C01820=1061.242,135.759,420.443,172.181,30.453,155.636
C01821=1061.248,136.008,420.422,172.183,30.455,155.637
C01822=1061.253,136.258,420.401,172.185,30.458,155.637
C01823=1061.259,136.507,420.381,172.186,30.461,155.638
C01824=1061.266,136.756,420.359,172.188,30.463,155.638
C01825=1061.271,137.005,420.339,172.190,30.466,155.638
C01826=1061.278,137.254,420.318,172.192,30.469,155.639
C01827=1061.283,137.503,420.297,172.193,30.471,155.639
C01828=1061.289,137.751,420.276,172.195,30.474,155.640
C01829=1061.295,138.001,420.255,172.197,30.477,155.640
C01830=1061.300,138.250,420.235,172.199,30.480,155.640
C01831=1061.307,138.499,420.213,172.201,30.482,155.641
C01832=1061.313,138.748,420.193,172.202,30.485,155.641
C01833=1061.319,138.997,420.172,172.204,30.488,155.642
C01834=1061.324,139.246,420.151,172.205,30.490,155.642
C01835=1061.331,139.495,420.130,172.207,30.493,155.643
C01836=1061.336,139.744,420.109,172.208,30.495,155.643
C01837=1061.342,139.993,420.088,172.210,30.498,155.643
C01838=1061.348,140.243,420.067,172.212,30.501,155.644
C01839=1061.353,140.491,420.046,172.214,30.503,155.644
C01840=1061.360,140.741,420.026,172.215,30.507,155.645
C01841=1061.365,140.989,420.004,172.217,30.509,155.645
C01842=1061.371,141.239,419.983,172.219,30.512,155.646
C01843=1061.377,141.488,419.962,172.221,30.515,155.646
C01844=1061.383,141.737,419.941,172.223,30.517,155.646
C01845=1061.388,141.986,419.920,172.224,30.520,155.647
C01846=1061.395,142.270,419.896,172.226,30.523,155.647
C01847=1061.402,142.554,419.872,172.229,30.526,155.648
C01848=1061.409,142.839,419.848,172.231,30.529,155.648
C01849=1061.416,143.123,419.824,172.232,30.533,155.649
C01850=1061.421,143.372,419.803,172.234,30.535,155.649
C01851=1061.427,143.621,419.781,172.236,30.538,155.650
C01852=1061.433,143.870,419.760,172.238,30.541,155.650
C01853=1061.438,144.120,419.739,172.239,30.543,155.650
C01854=1061.444,144.368,419.718,172.241,30.546,155.651
C01855=1061.450,144.617,419.696,172.243,30.549,155.651
C01856=1061.455,144.866,419.676,172.245,30.551,155.652
C01857=1061.462,145.115,419.655,172.246,30.554,155.652
C01858=1061.468,145.364,419.633,172.248,30.557,155.653
C01859=1061.474,145.613,419.612,172.250,30.560,155.653
C01860=1061.480,145.863,419.591,172.252,30.563,155.653
C01861=1061.486,146.111,419.570,172.254,30.565,155.654
C01862=1061.492,146.361,419.548,172.255,30.568,155.654
C01863=1061.497,146.610,419.527,172.257,30.571,155.655
C01864=1061.503,146.859,419.506,172.259,30.573,155.655
C01865=1061.509,147.107,419.485,172.261,30.576,155.655
C01866=1061.515,147.357,419.463,172.262,30.579,155.656
C01867=1061.522,147.605,419.442,172.264,30.581,155.656
C01868=1061.527,147.855,419.421,172.266,30.584,155.657
C01869=1061.532,148.104,419.399,172.268,30.587,155.657
C01870=1061.538,148.353,419.378,172.270,30.590,155.658
C01871=1061.544,148.602,419.356,172.271,30.592,155.658
C01872=1061.550,148.850,419.335,172.273,30.595,155.658
C01873=1061.556,149.100,419.313,172.275,30.598,155.659
C01874=1061.562,149.349,419.292,172.277,30.600,155.659
C01875=1061.567,149.598,419.271,172.278,30.603,155.660
C01876=1061.573,149.847,419.249,172.280,30.606,155.660
C01877=1061.579,150.096,419.228,172.282,30.609,155.661
C01878=1061.585,150.345,419.207,172.284,30.612,155.661
C01879=1061.591,150.594,419.185,172.286,30.614,155.662
C01880=1061.597,150.843,419.164,172.287,30.617,155.662
C01881=1061.603,151.092,419.142,172.289,30.620,155.662
C01882=1061.608,151.341,419.120,172.291,30.622,155.663
C01883=1061.614,151.590,419.099,172.294,30.625,155.663
C01884=1061.620,151.839,419.077,172.295,30.628,155.664
C01885=1061.626,152.087,419.056,172.297,30.631,155.664
C01886=1061.632,152.337,419.034,172.299,30.634,155.665
C01887=1061.637,152.585,419.013,172.301,30.636,155.665
C01888=1061.644,152.834,418.991,172.302,30.639,155.665
C01889=1061.649,153.084,418.969,172.304,30.642,155.666
C01890=1061.655,153.332,418.948,172.306,30.645,155.666
C01891=1061.661,153.582,418.926,172.308,30.648,155.667
C01892=1061.667,153.831,418.904,172.310,30.650,155.667
C01893=1061.673,154.079,418.883,172.311,30.653,155.668
C01894=1061.679,154.329,418.861,172.313,30.656,155.668
C01895=1061.684,154.578,418.839,172.315,30.658,155.668
C01896=1061.690,154.827,418.818,172.317,30.661,155.669
C01897=1061.696,155.076,418.796,172.318,30.664,155.669
C01898=1061.702,155.325,418.775,172.320,30.667,155.670
C01899=1061.708,155.573,418.753,172.322,30.669,155.670
C01900=1061.713,155.822,418.730,172.324,30.672,155.671
C01901=1061.719,156.072,418.709,172.326,30.675,155.671
C01902=1061.726,156.321,418.687,172.327,30.678,155.671
C01903=1061.730,156.570,418.665,172.330,30.681,155.672
C01904=1061.737,156.819,418.644,172.332,30.684,155.672
C01905=1061.743,157.068,418.622,172.334,30.686,155.673
C01906=1061.748,157.316,418.599,172.336,30.689,155.673
C01907=1061.754,157.565,418.578,172.337,30.692,155.674
C01908=1061.760,157.815,418.556,172.339,30.695,155.674
C01909=1061.766,158.063,418.535,172.341,30.697,155.675
C01910=1061.773,158.348,418.509,172.343,30.701,155.675
C01911=1061.779,158.631,418.484,172.345,30.704,155.676
C01912=1061.786,158.915,418.460,172.347,30.707,155.676
C01913=1061.793,159.200,418.434,172.349,30.710,155.676
C01914=1061.798,159.448,418.413,172.351,30.713,155.677
C01915=1061.804,159.698,418.391,172.353,30.716,155.677
C01916=1061.810,159.946,418.368,172.355,30.719,155.678
C01917=1061.816,160.196,418.347,172.357,30.721,155.678
C01918=1061.821,160.444,418.325,172.359,30.724,155.679
C01919=1061.827,160.693,418.303,172.361,30.727,155.679
C01920=1061.834,160.942,418.281,172.362,30.729,155.679
C01921=1061.839,161.192,418.259,172.364,30.732,155.680
C01922=1061.845,161.440,418.237,172.366,30.735,155.680
C01923=1061.850,161.689,418.214,172.368,30.738,155.681
C01924=1061.856,161.938,418.191,172.369,30.741,155.681
C01925=1061.862,162.187,418.170,172.371,30.744,155.682
C01926=1061.867,162.436,418.148,172.374,30.747,155.682
C01927=1061.873,162.685,418.125,172.376,30.750,155.683
C01928=1061.879,162.934,418.103,172.378,30.752,155.683
C01929=1061.884,163.182,418.081,172.379,30.756,155.684
C01930=1061.889,163.432,418.059,172.381,30.758,155.684
C01931=1061.896,163.680,418.036,172.383,30.761,155.685
C01932=1061.901,163.930,418.014,172.385,30.764,155.685
C01933=1061.907,164.178,417.991,172.386,30.767,155.685
C01934=1061.913,164.427,417.970,172.388,30.770,155.686
C01935=1061.918,164.676,417.947,172.390,30.773,155.686
C01936=1061.924,164.926,417.925,172.393,30.775,155.687
C01937=1061.929,165.174,417.902,172.395,30.779,155.687
C01938=1061.935,165.423,417.880,172.396,30.781,155.688
C01939=1061.941,165.672,417.857,172.398,30.785,155.688
C01940=1061.946,165.922,417.835,172.400,30.787,155.689
C01941=1061.952,166.169,417.813,172.402,30.790,155.689
C01942=1061.958,166.419,417.791,172.403,30.793,155.690
C01943=1061.963,166.668,417.768,172.405,30.796,155.690
C01944=1061.970,166.916,417.746,172.407,30.798,155.691
C01945=1061.975,167.166,417.723,172.410,30.802,155.691
C01946=1061.981,167.415,417.701,172.412,30.804,155.691
C01947=1061.986,167.664,417.679,172.413,30.808,155.692
C01948=1061.992,167.912,417.656,172.415,30.810,155.692
C01949=1061.998,168.161,417.633,172.417,30.813,155.693
C01950=1062.003,168.411,417.611,172.419,30.816,155.693
C01951=1062.009,168.660,417.588,172.421,30.819,155.694
C01952=1062.016,168.908,417.566,172.423,30.822,155.694
C01953=1062.020,169.157,417.544,172.425,30.825,155.695
C01954=1062.026,169.406,417.521,172.427,30.827,155.695
C01955=1062.033,169.654,417.499,172.429,30.830,155.696
C01956=1062.038,169.904,417.476,172.430,30.833,155.696
C01957=1062.044,170.153,417.454,172.432,30.836,155.696
C01958=1062.049,170.402,417.431,172.434,30.839,155.697
C01959=1062.055,170.651,417.408,172.437,30.842,155.697
C01960=1062.061,170.900,417.386,172.439,30.845,155.698
C01961=1062.067,171.148,417.363,172.440,30.848,155.698
C01962=1062.072,171.397,417.340,172.442,30.850,155.699
C01963=1062.078,171.646,417.318,172.444,30.853,155.699
C01964=1062.084,171.895,417.296,172.446,30.856,155.700
C01965=1062.090,172.144,417.273,172.448,30.859,155.700
C01966=1062.096,172.393,417.250,172.450,30.862,155.701
C01967=1062.101,172.642,417.227,172.452,30.865,155.701
C01968=1062.108,172.890,417.205,172.454,30.868,155.702
C01969=1062.113,173.140,417.182,172.456,30.871,155.702
C01970=1062.119,173.389,417.160,172.457,30.874,155.702
C01971=1062.125,173.638,417.137,172.460,30.876,155.703
C01972=1062.130,173.887,417.114,172.462,30.880,155.703
C01973=1062.137,174.135,417.091,172.464,30.882,155.704
C01974=1062.143,174.419,417.066,172.467,30.886,155.704
C01975=1062.150,174.703,417.040,172.468,30.889,155.705
C01976=1062.156,174.986,417.013,172.471,30.892,155.705
C01977=1062.163,175.270,416.988,172.473,30.895,155.706
C01978=1062.169,175.518,416.965,172.475,30.898,155.706
C01979=1062.175,175.767,416.942,172.476,30.901,155.707
C01980=1062.180,176.016,416.919,172.479,30.904,155.707
C01981=1062.186,176.265,416.896,172.481,30.907,155.708
C01982=1062.192,176.514,416.874,172.483,30.910,155.708
C01983=1062.198,176.763,416.851,172.485,30.912,155.709
C01984=1062.204,177.012,416.828,172.486,30.915,155.709
C01985=1062.210,177.261,416.805,172.489,30.919,155.710
C01986=1062.216,177.510,416.782,172.491,30.921,155.710
C01987=1062.222,177.759,416.759,172.493,30.924,155.710
C01988=1062.228,178.008,416.736,172.495,30.927,155.711
C01989=1062.233,178.257,416.713,172.497,30.930,155.711
C01990=1062.240,178.505,416.691,172.499,30.932,155.712
C01991=1062.246,178.754,416.668,172.501,30.936,155.712
C01992=1062.251,179.003,416.645,172.503,30.938,155.713
C01993=1062.257,179.252,416.622,172.505,30.941,155.713
C01994=1062.263,179.501,416.599,172.507,30.944,155.714
C01995=1062.269,179.749,416.575,172.509,30.947,155.714
C01996=1062.275,179.998,416.553,172.511,30.950,155.715
C01997=1062.282,180.247,416.530,172.513,30.953,155.715
C01998=1062.287,180.496,416.507,172.516,30.956,155.715
C01999=1062.293,180.745,416.484,172.517,30.959,155.716
C02000=1062.299,180.994,416.461,172.519,30.961,155.716
C02001=1062.305,181.243,416.438,172.521,30.964,155.717
C02002=1062.311,181.491,416.414,172.524,30.967,155.717
C02003=1062.316,181.740,416.391,172.525,30.970,155.718
C02004=1062.323,181.989,416.369,172.527,30.973,155.718
C02005=1062.329,182.238,416.346,172.529,30.976,155.719
C02006=1062.335,182.487,416.323,172.532,30.979,155.719
C02007=1062.341,182.735,416.299,172.534,30.981,155.720
C02008=1062.347,182.984,416.276,172.535,30.984,155.720
C02009=1062.353,183.234,416.253,172.538,30.987,155.720
C02010=1062.359,183.483,416.230,172.540,30.990,155.721
C02011=1062.364,183.732,416.207,172.542,30.993,155.721
C02012=1062.370,183.980,416.183,172.544,30.996,155.722
C02013=1062.376,184.229,416.160,172.546,30.999,155.722
C02014=1062.383,184.478,416.138,172.548,31.002,155.723
C02015=1062.389,184.727,416.113,172.550,31.005,155.723
C02016=1062.394,184.976,416.090,172.552,31.008,155.724
C02017=1062.399,185.225,416.067,172.555,31.011,155.724
C02018=1062.405,185.473,416.043,172.556,31.014,155.725
C02019=1062.411,185.722,416.020,172.558,31.017,155.725
C02020=1062.416,185.971,415.996,172.561,31.020,155.726
C02021=1062.422,186.220,415.973,172.563,31.023,155.726
C02022=1062.428,186.469,415.950,172.565,31.026,155.727
C02023=1062.434,186.718,415.925,172.566,31.029,155.727
C02024=1062.439,186.967,415.902,172.569,31.032,155.728
C02025=1062.445,187.215,415.879,172.571,31.035,155.728
C02026=1062.450,187.464,415.855,172.573,31.038,155.729
C02027=1062.456,187.712,415.832,172.575,31.041,155.729
C02028=1062.461,187.962,415.808,172.577,31.044,155.730
C02029=1062.468,188.211,415.784,172.579,31.048,155.730
C02030=1062.474,188.459,415.761,172.581,31.050,155.731
C02031=1062.479,188.708,415.737,172.584,31.053,155.731
C02032=1062.485,188.957,415.714,172.585,31.057,155.732
C02033=1062.490,189.206,415.690,172.587,31.059,155.732
C02034=1062.496,189.454,415.667,172.590,31.063,155.733
C02035=1062.503,189.703,415.643,172.592,31.066,155.733
C02036=1062.508,189.952,415.618,172.594,31.068,155.734
C02037=1062.514,190.201,415.595,172.595,31.072,155.734
C02038=1062.520,190.484,415.568,172.598,31.075,155.735
C02039=1062.527,190.768,415.542,172.601,31.079,155.735
C02040=1062.533,191.050,415.514,172.603,31.082,155.736
C02041=1062.540,191.334,415.487,172.606,31.086,155.736
C02042=1062.546,191.583,415.464,172.607,31.089,155.737
C02043=1062.551,191.831,415.439,172.610,31.091,155.737
C02044=1062.557,192.080,415.416,172.612,31.095,155.738
C02045=1062.563,192.329,415.392,172.614,31.098,155.738
C02046=1062.569,192.578,415.368,172.617,31.101,155.739
C02047=1062.575,192.826,415.345,172.618,31.104,155.739
C02048=1062.580,193.075,415.321,172.620,31.107,155.740
C02049=1062.586,193.324,415.297,172.623,31.110,155.740
C02050=1062.591,193.573,415.273,172.625,31.113,155.741
C02051=1062.597,193.822,415.250,172.627,31.116,155.741
C02052=1062.603,194.071,415.225,172.629,31.120,155.742
C02053=1062.609,194.319,415.202,172.631,31.122,155.742
C02054=1062.615,194.568,415.178,172.633,31.125,155.743
C02055=1062.621,194.817,415.153,172.636,31.129,155.743
C02056=1062.627,195.066,415.130,172.638,31.131,155.744
C02057=1062.632,195.314,415.106,172.639,31.135,155.744
C02058=1062.639,195.563,415.082,172.642,31.138,155.745
C02059=1062.644,195.812,415.058,172.644,31.140,155.745
C02060=1062.650,196.060,415.034,172.647,31.144,155.746
C02061=1062.656,196.310,415.010,172.649,31.147,155.746
C02062=1062.662,196.558,414.987,172.650,31.150,155.747
C02063=1062.668,196.808,414.962,172.653,31.153,155.747
C02064=1062.674,197.056,414.938,172.655,31.156,155.748
C02065=1062.679,197.305,414.914,172.657,31.159,155.748
C02066=1062.686,197.554,414.890,172.660,31.162,155.749
C02067=1062.691,197.802,414.866,172.661,31.165,155.749
C02068=1062.697,198.050,414.842,172.664,31.169,155.750
C02069=1062.703,198.300,414.817,172.666,31.171,155.750
C02070=1062.709,198.548,414.794,172.668,31.174,155.751
C02071=1062.714,198.798,414.770,172.671,31.178,155.751
C02072=1062.720,199.046,414.746,172.672,31.180,155.752
C02073=1062.726,199.295,414.722,172.675,31.184,155.752
C02074=1062.732,199.544,414.698,172.677,31.187,155.753
C02075=1062.738,199.793,414.673,172.679,31.190,155.753
C02076=1062.744,200.041,414.650,172.682,31.193,155.754
C02077=1062.750,200.290,414.625,172.683,31.196,155.754
C02078=1062.756,200.539,414.601,172.686,31.199,155.755
C02079=1062.762,200.787,414.576,172.688,31.202,155.755
C02080=1062.768,201.036,414.552,172.690,31.205,155.756
C02081=1062.774,201.284,414.528,172.693,31.209,155.756
C02082=1062.780,201.534,414.503,172.694,31.211,155.757
C02083=1062.786,201.782,414.480,172.697,31.214,155.757
C02084=1062.792,202.031,414.455,172.699,31.218,155.758
C02085=1062.797,202.280,414.431,172.702,31.221,155.758
C02086=1062.804,202.529,414.407,172.704,31.224,155.759
C02087=1062.809,202.777,414.383,172.705,31.227,155.759
C02088=1062.815,203.026,414.357,172.708,31.230,155.760
C02089=1062.820,203.275,414.333,172.710,31.233,155.760
C02090=1062.826,203.524,414.308,172.713,31.237,155.761
C02091=1062.832,203.772,414.285,172.715,31.240,155.761
C02092=1062.838,204.021,414.260,172.717,31.243,155.762
C02093=1062.844,204.269,414.235,172.719,31.246,155.763
C02094=1062.850,204.519,414.211,172.721,31.250,155.763
C02095=1062.855,204.767,414.186,172.724,31.253,155.764
C02096=1062.861,205.017,414.162,172.726,31.256,155.764
C02097=1062.867,205.264,414.137,172.728,31.259,155.765
C02098=1062.873,205.514,414.113,172.730,31.262,155.765
C02099=1062.879,205.762,414.088,172.733,31.265,155.766
C02100=1062.884,206.011,414.064,172.735,31.268,155.766
C02101=1062.890,206.259,414.039,172.738,31.272,155.767
C02102=1062.915,207.308,413.935,172.906,31.353,155.774
C02103=1062.920,207.532,413.912,172.908,31.357,155.775
C02104=1062.926,207.757,413.890,172.910,31.361,155.775
C02105=1062.931,207.982,413.866,172.911,31.364,155.776
C02106=1062.937,208.207,413.844,172.913,31.368,155.777
C02107=1062.943,208.432,413.821,172.915,31.372,155.777
C02108=1062.948,208.657,413.797,172.917,31.376,155.778
C02109=1062.953,208.881,413.775,172.919,31.379,155.779
C02110=1062.959,209.107,413.752,172.920,31.383,155.779
C02111=1062.965,209.355,413.726,172.922,31.387,155.780
C02112=1062.971,209.604,413.700,172.924,31.391,155.781
C02113=1062.977,209.852,413.674,172.926,31.395,155.782
C02114=1062.983,210.101,413.649,172.928,31.399,155.782
C02115=1062.989,210.350,413.624,172.930,31.404,155.783
C02116=1062.996,210.598,413.598,172.932,31.407,155.784
C02117=1063.001,210.847,413.572,172.934,31.412,155.784
C02118=1063.008,211.095,413.546,172.936,31.415,155.785
C02119=1063.014,211.344,413.521,172.937,31.420,155.786
C02120=1063.019,211.593,413.495,172.939,31.423,155.787
C02121=1063.025,211.842,413.470,172.942,31.428,155.787
C02122=1063.032,212.090,413.444,172.944,31.432,155.788
C02123=1063.038,212.338,413.418,172.946,31.436,155.789
C02124=1063.044,212.587,413.392,172.947,31.440,155.790
C02125=1063.050,212.836,413.367,172.949,31.444,155.790
C02126=1063.055,213.085,413.341,172.952,31.448,155.791
C02127=1063.062,213.333,413.315,172.954,31.452,155.792
C02128=1063.068,213.582,413.290,172.956,31.456,155.792
C02129=1063.073,213.831,413.264,172.957,31.460,155.793
C02130=1063.080,214.079,413.238,172.959,31.464,155.794
C02131=1063.085,214.328,413.212,172.962,31.469,155.795
C02132=1063.092,214.576,413.186,172.964,31.472,155.795
C02133=1063.097,214.825,413.160,172.966,31.477,155.796
C02134=1063.104,215.073,413.134,172.967,31.480,155.797
C02135=1063.109,215.322,413.108,172.969,31.485,155.798
C02136=1063.116,215.570,413.082,172.972,31.488,155.798
C02137=1063.122,215.819,413.057,172.974,31.493,155.799
C02138=1063.128,216.068,413.031,172.976,31.496,155.800
C02139=1063.134,216.316,413.005,172.977,31.501,155.801
C02140=1063.140,216.565,412.979,172.979,31.504,155.801
C02141=1063.146,216.813,412.953,172.982,31.509,155.802
C02142=1063.152,217.062,412.927,172.984,31.513,155.803
C02143=1063.158,217.310,412.901,172.986,31.517,155.803
C02144=1063.164,217.559,412.875,172.987,31.521,155.804
C02145=1063.170,217.808,412.849,172.990,31.525,155.805
C02146=1063.176,218.056,412.822,172.992,31.529,155.806
C02147=1063.182,218.305,412.797,172.994,31.533,155.806
C02148=1063.188,218.553,412.770,172.996,31.537,155.807
C02149=1063.194,218.802,412.745,172.998,31.541,155.808
C02150=1063.200,219.050,412.718,173.000,31.545,155.808
C02151=1063.206,219.299,412.693,173.002,31.549,155.809
C02152=1063.212,219.547,412.666,173.004,31.553,155.810
C02153=1063.219,219.797,412.641,173.007,31.557,155.811
C02154=1063.225,220.045,412.614,173.008,31.561,155.811
C02155=1063.231,220.293,412.588,173.010,31.565,155.812
C02156=1063.237,220.542,412.562,173.012,31.569,155.813
C02157=1063.243,220.790,412.536,173.015,31.573,155.813
C02158=1063.249,221.039,412.509,173.017,31.577,155.814
C02159=1063.254,221.266,412.485,173.019,31.581,155.815
C02160=1063.260,221.494,412.461,173.020,31.584,155.815
C02161=1063.265,221.721,412.438,173.022,31.588,155.816
C02162=1063.271,221.948,412.413,173.024,31.591,155.817
C02163=1063.277,222.176,412.389,173.026,31.595,155.817
C02164=1063.282,222.403,412.365,173.028,31.599,155.818
C02165=1063.288,222.630,412.341,173.030,31.602,155.819
C02166=1063.293,222.858,412.317,173.031,31.606,155.820
C02167=1063.299,223.106,412.290,173.034,31.611,155.820
C02168=1063.305,223.355,412.264,173.036,31.614,155.821
C02169=1063.310,223.603,412.237,173.038,31.619,155.822
C02170=1063.318,223.852,412.211,173.041,31.622,155.822
C02171=1063.323,224.100,412.184,173.042,31.627,155.823
C02172=1063.329,224.349,412.158,173.044,31.630,155.824
C02173=1063.335,224.598,412.132,173.046,31.635,155.825
C02174=1063.341,224.846,412.106,173.049,31.638,155.825
C02175=1063.347,225.095,412.079,173.051,31.642,155.826
C02176=1063.353,225.343,412.052,173.053,31.646,155.827
C02177=1063.359,225.592,412.025,173.055,31.650,155.827
C02178=1063.365,225.840,411.999,173.057,31.655,155.828
C02179=1063.372,226.089,411.972,173.059,31.658,155.829
C02180=1063.378,226.337,411.946,173.061,31.662,155.830
C02181=1063.383,226.585,411.919,173.064,31.666,155.830
C02182=1063.389,226.834,411.892,173.066,31.670,155.831
C02183=1063.395,227.084,411.866,173.067,31.674,155.832
C02184=1063.402,227.332,411.840,173.070,31.678,155.832
C02185=1063.408,227.580,411.813,173.072,31.682,155.833
C02186=1063.414,227.829,411.786,173.074,31.686,155.834
C02187=1063.420,228.077,411.760,173.077,31.690,155.835
C02188=1063.425,228.326,411.733,173.078,31.694,155.835
C02189=1063.433,228.574,411.707,173.080,31.698,155.836
C02190=1063.439,228.822,411.679,173.083,31.702,155.837
C02191=1063.444,229.071,411.653,173.085,31.706,155.838
C02192=1063.451,229.320,411.626,173.087,31.710,155.838
C02193=1063.457,229.568,411.599,173.090,31.714,155.839
C02194=1063.462,229.816,411.572,173.091,31.718,155.840
C02195=1063.469,230.065,411.545,173.093,31.721,155.840
C02196=1063.475,230.314,411.519,173.096,31.726,155.841
C02197=1063.480,230.562,411.492,173.098,31.730,155.842
C02198=1063.487,230.811,411.465,173.100,31.734,155.843
C02199=1063.492,231.060,411.438,173.103,31.738,155.843
C02200=1063.499,231.307,411.411,173.104,31.742,155.844
C02201=1063.505,231.556,411.384,173.106,31.746,155.845
C02202=1063.511,231.805,411.357,173.109,31.749,155.845
C02203=1063.516,232.053,411.331,173.111,31.754,155.846
C02204=1063.523,232.302,411.304,173.113,31.757,155.847
C02205=1063.529,232.550,411.276,173.116,31.762,155.848
C02206=1063.535,232.798,411.250,173.117,31.765,155.848
C02207=1063.541,233.047,411.223,173.119,31.770,155.849
C02208=1063.547,233.296,411.196,173.122,31.774,155.850
C02209=1063.553,233.544,411.168,173.124,31.777,155.850
C02210=1063.559,233.792,411.142,173.127,31.782,155.851
C02211=1063.564,234.041,411.114,173.129,31.785,155.852
C02212=1063.571,234.290,411.087,173.131,31.790,155.853
C02213=1063.577,234.538,411.060,173.133,31.793,155.853
C02214=1063.583,234.786,411.033,173.135,31.798,155.854
C02215=1063.588,235.010,411.009,173.137,31.801,155.855
C02216=1063.594,235.233,410.984,173.139,31.804,155.855
C02217=1063.599,235.457,410.960,173.141,31.808,155.856
C02218=1063.605,235.680,410.936,173.144,31.812,155.857
C02219=1063.610,235.903,410.911,173.146,31.815,155.857
C02220=1063.616,236.127,410.887,173.147,31.819,155.858
C02221=1063.621,236.350,410.862,173.149,31.822,155.859
C02222=1063.626,236.574,410.837,173.151,31.826,155.859
C02223=1063.632,236.821,410.810,173.154,31.830,155.860
C02224=1063.638,237.070,410.783,173.156,31.834,155.861
C02225=1063.644,237.318,410.756,173.158,31.838,155.861
C02226=1063.651,237.567,410.729,173.160,31.842,155.862
C02227=1063.657,237.815,410.701,173.162,31.846,155.863
C02228=1063.662,238.064,410.674,173.165,31.850,155.864
C02229=1063.669,238.312,410.646,173.167,31.853,155.864
C02230=1063.675,238.561,410.619,173.169,31.858,155.865
C02231=1063.681,238.809,410.592,173.172,31.861,155.866
C02232=1063.687,239.058,410.563,173.174,31.865,155.866
C02233=1063.693,239.306,410.537,173.176,31.869,155.867
C02234=1063.699,239.554,410.509,173.178,31.873,155.868
C02235=1063.705,239.803,410.482,173.180,31.877,155.868
C02236=1063.711,240.052,410.454,173.183,31.881,155.869
C02237=1063.717,240.299,410.427,173.185,31.885,155.870
C02238=1063.724,240.548,410.400,173.188,31.889,155.871
C02239=1063.729,240.796,410.372,173.190,31.893,155.871
C02240=1063.736,241.045,410.344,173.192,31.897,155.872
C02241=1063.742,241.294,410.317,173.194,31.900,155.873
C02242=1063.748,241.542,410.290,173.197,31.905,155.874
C02243=1063.754,241.790,410.261,173.199,31.908,155.874
C02244=1063.760,242.039,410.235,173.201,31.912,155.875
C02245=1063.766,242.287,410.207,173.204,31.917,155.876
C02246=1063.772,242.535,410.179,173.206,31.920,155.876
C02247=1063.778,242.784,410.151,173.208,31.925,155.877
C02248=1063.784,243.033,410.124,173.210,31.928,155.878
C02249=1063.790,243.281,410.096,173.213,31.932,155.878
C02250=1063.796,243.530,410.068,173.215,31.936,155.879
C02251=1063.802,243.777,410.041,173.218,31.940,155.880
C02252=1063.808,244.026,410.012,173.220,31.944,155.881
C02253=1063.814,244.274,409.986,173.222,31.948,155.881
C02254=1063.820,244.523,409.957,173.224,31.952,155.882
C02255=1063.827,244.772,409.930,173.226,31.956,155.883
C02256=1063.832,245.020,409.902,173.229,31.960,155.884
C02257=1063.839,245.268,409.874,173.231,31.964,155.884
C02258=1063.844,245.516,409.846,173.234,31.968,155.885
C02259=1063.851,245.765,409.818,173.236,31.972,155.886
C02260=1063.857,246.013,409.790,173.239,31.976,155.886
C02261=1063.862,246.261,409.762,173.241,31.980,155.887
C02262=1063.869,246.510,409.734,173.243,31.984,155.888
C02263=1063.874,246.758,409.706,173.245,31.988,155.889
C02264=1063.880,247.007,409.678,173.248,31.992,155.889
C02265=1063.886,247.255,409.650,173.250,31.996,155.890
C02266=1063.892,247.503,409.622,173.253,32.000,155.891
C02267=1063.898,247.752,409.594,173.255,32.004,155.892
C02268=1063.904,248.000,409.567,173.257,32.007,155.892
C02269=1063.910,248.248,409.538,173.259,32.012,155.893
C02270=1063.916,248.497,409.510,173.261,32.015,155.894
C02271=1063.921,248.717,409.485,173.264,32.019,155.894
C02272=1063.926,248.937,409.460,173.266,32.023,155.895
C02273=1063.932,249.157,409.435,173.268,32.026,155.896
C02274=1063.937,249.378,409.410,173.270,32.030,155.896
C02275=1063.942,249.598,409.386,173.272,32.033,155.897
C02276=1063.947,249.818,409.360,173.275,32.037,155.898
C02277=1063.953,250.038,409.336,173.277,32.040,155.898
C02278=1063.957,250.259,409.311,173.278,32.044,155.899
C02279=1063.964,250.507,409.282,173.281,32.048,155.900
C02280=1063.970,250.755,409.254,173.283,32.052,155.900
C02281=1063.976,251.003,409.226,173.286,32.056,155.901
C02282=1063.982,251.252,409.198,173.288,32.060,155.902
C02283=1063.988,251.500,409.168,173.291,32.064,155.902
C02284=1063.993,251.748,409.141,173.293,32.068,155.903
C02285=1064.000,251.997,409.113,173.296,32.072,155.904
C02286=1064.006,252.246,409.084,173.297,32.076,155.905
C02287=1064.012,252.493,409.056,173.300,32.080,155.905
C02288=1064.017,252.742,409.027,173.302,32.083,155.906
C02289=1064.023,252.991,408.999,173.305,32.088,155.907
C02290=1064.030,253.238,408.971,173.307,32.091,155.908
C02291=1064.036,253.487,408.942,173.310,32.096,155.908
C02292=1064.042,253.735,408.914,173.312,32.099,155.909
C02293=1064.048,253.983,408.885,173.315,32.103,155.910
C02294=1064.054,254.232,408.857,173.317,32.107,155.911
C02295=1064.060,254.481,408.829,173.319,32.111,155.911
C02296=1064.066,254.728,408.801,173.322,32.115,155.912
C02297=1064.072,254.977,408.772,173.324,32.119,155.913
C02298=1064.078,255.225,408.743,173.327,32.123,155.913
C02299=1064.084,255.474,408.715,173.329,32.127,155.914
C02300=1064.091,255.722,408.686,173.332,32.131,155.915
C02301=1064.097,255.970,408.658,173.335,32.135,155.915
C02302=1064.102,256.218,408.629,173.337,32.139,155.916
C02303=1064.109,256.466,408.601,173.339,32.143,155.917
C02304=1064.115,256.714,408.572,173.341,32.146,155.918
C02305=1064.121,256.963,408.544,173.344,32.151,155.918
C02306=1064.127,257.211,408.515,173.346,32.154,155.919
C02307=1064.133,257.460,408.486,173.349,32.158,155.920
C02308=1064.140,257.708,408.457,173.352,32.162,155.921
C02309=1064.145,257.957,408.429,173.354,32.166,155.921
C02310=1064.151,258.204,408.400,173.357,32.170,155.922
C02311=1064.158,258.453,408.373,173.359,32.174,155.923
C02312=1064.164,258.701,408.344,173.361,32.178,155.923
C02313=1064.170,258.949,408.315,173.364,32.181,155.924
C02314=1064.176,259.198,408.286,173.366,32.186,155.925
C02315=1064.182,259.446,408.257,173.369,32.189,155.926
C02316=1064.189,259.694,408.228,173.371,32.193,155.926
C02317=1064.195,259.943,408.200,173.374,32.197,155.927
C02318=1064.201,260.191,408.171,173.377,32.201,155.928
C02319=1064.207,260.439,408.142,173.379,32.205,155.928
C02320=1064.213,260.688,408.113,173.382,32.209,155.929
C02321=1064.220,260.936,408.085,173.384,32.213,155.930
C02322=1064.226,261.184,408.056,173.386,32.217,155.931
C02323=1064.233,261.432,408.027,173.389,32.220,155.931
C02324=1064.239,261.681,407.999,173.391,32.225,155.932
C02325=1064.245,261.929,407.970,173.394,32.228,155.933
C02326=1064.251,262.177,407.941,173.397,32.232,155.933
C02327=1064.257,262.397,407.915,173.399,32.236,155.934
C02328=1064.262,262.615,407.889,173.401,32.239,155.935
C02329=1064.267,262.835,407.864,173.404,32.243,155.935
C02330=1064.273,263.053,407.839,173.406,32.246,155.936
C02331=1064.278,263.273,407.813,173.408,32.249,155.937
C02332=1064.284,263.492,407.787,173.410,32.252,155.937
C02333=1064.289,263.711,407.762,173.412,32.256,155.938
C02334=1064.295,263.930,407.736,173.414,32.260,155.938
C02335=1064.301,264.178,407.707,173.417,32.263,155.939
C02336=1064.307,264.426,407.678,173.420,32.268,155.940
C02337=1064.313,264.675,407.648,173.422,32.271,155.941
C02338=1064.319,264.923,407.619,173.425,32.276,155.941
C02339=1064.325,265.171,407.590,173.428,32.280,155.942
C02340=1064.332,265.419,407.561,173.430,32.283,155.943
C02341=1064.337,265.668,407.531,173.433,32.287,155.944
C02342=1064.343,265.916,407.502,173.436,32.291,155.944
C02343=1064.350,266.164,407.473,173.437,32.295,155.945
C02344=1064.356,266.412,407.444,173.440,32.299,155.946
C02345=1064.361,266.660,407.414,173.443,32.303,155.946
C02346=1064.368,266.908,407.385,173.445,32.307,155.947
C02347=1064.374,267.157,407.356,173.448,32.311,155.948
C02348=1064.379,267.405,407.327,173.451,32.315,155.949
C02349=1064.386,267.653,407.298,173.453,32.319,155.949
C02350=1064.392,267.901,407.269,173.456,32.323,155.950
C02351=1064.398,268.149,407.238,173.459,32.327,155.951
C02352=1064.404,268.397,407.209,173.461,32.331,155.952
C02353=1064.410,268.645,407.180,173.464,32.335,155.952
C02354=1064.417,268.894,407.151,173.466,32.339,155.953
C02355=1064.422,269.143,407.121,173.468,32.343,155.954
C02356=1064.429,269.391,407.092,173.471,32.347,155.954
C02357=1064.435,269.639,407.062,173.474,32.351,155.955
C02358=1064.441,269.887,407.033,173.476,32.354,155.956
C02359=1064.446,270.135,407.003,173.479,32.359,155.957
C02360=1064.453,270.383,406.973,173.482,32.363,155.957
C02361=1064.459,270.631,406.944,173.485,32.367,155.958
C02362=1064.465,270.879,406.915,173.487,32.370,155.959
C02363=1064.472,271.128,406.885,173.490,32.375,155.960
C02364=1064.477,271.376,406.855,173.493,32.378,155.960
C02365=1064.484,271.624,406.826,173.495,32.382,155.961
C02366=1064.489,271.872,406.796,173.497,32.386,155.962
C02367=1064.496,272.120,406.767,173.500,32.390,155.963
C02368=1064.501,272.368,406.737,173.503,32.394,155.963
C02369=1064.508,272.617,406.707,173.505,32.398,155.964
C02370=1064.514,272.865,406.677,173.508,32.402,155.965
C02371=1064.520,273.113,406.647,173.511,32.406,155.965
C02372=1064.526,273.361,406.618,173.513,32.410,155.966
C02373=1064.532,273.609,406.588,173.516,32.414,155.967
C02374=1064.538,273.857,406.558,173.519,32.418,155.968
C02375=1064.545,274.105,406.528,173.522,32.422,155.968
C02376=1064.551,274.354,406.499,173.524,32.426,155.969
C02377=1064.556,274.602,406.468,173.527,32.430,155.970
C02378=1064.563,274.850,406.439,173.530,32.434,155.971
C02379=1064.568,275.097,406.409,173.532,32.438,155.971
C02380=1064.575,275.347,406.379,173.534,32.442,155.972
C02381=1064.581,275.594,406.349,173.537,32.446,155.973
C02382=1064.587,275.842,406.319,173.540,32.450,155.974
C02383=1064.593,276.063,406.293,173.542,32.454,155.974
C02384=1064.598,276.284,406.266,173.545,32.458,155.975
C02385=1064.603,276.505,406.239,173.547,32.461,155.976
C02386=1064.609,276.726,406.213,173.550,32.464,155.976
C02387=1064.614,276.947,406.186,173.552,32.468,155.977
C02388=1064.620,277.168,406.158,173.555,32.472,155.978
C02389=1064.625,277.388,406.132,173.557,32.475,155.978
C02390=1064.630,277.609,406.105,173.560,32.479,155.979
C02391=1064.637,277.858,406.075,173.562,32.483,155.980
C02392=1064.643,278.106,406.046,173.565,32.487,155.981
C02393=1064.649,278.354,406.015,173.568,32.491,155.981
C02394=1064.655,278.602,405.985,173.570,32.495,155.982
C02395=1064.662,278.850,405.955,173.572,32.499,155.983
C02396=1064.667,279.098,405.925,173.575,32.503,155.983
C02397=1064.674,279.347,405.894,173.578,32.507,155.984
C02398=1064.679,279.595,405.864,173.581,32.511,155.985
C02399=1064.686,279.842,405.834,173.584,32.515,155.986
C02400=1064.692,280.091,405.804,173.586,32.519,155.986
C02401=1064.698,280.338,405.773,173.589,32.523,155.987
C02402=1064.704,280.586,405.743,173.592,32.527,155.988
C02403=1064.710,280.835,405.713,173.595,32.531,155.989
C02404=1064.716,281.083,405.683,173.598,32.535,155.989
C02405=1064.722,281.331,405.652,173.600,32.539,155.990
C02406=1064.728,281.580,405.621,173.603,32.543,155.991
C02407=1064.735,281.827,405.592,173.606,32.547,155.992
C02408=1064.741,282.075,405.561,173.609,32.551,155.993
C02409=1064.747,282.323,405.531,173.612,32.556,155.993
C02410=1064.753,282.571,405.500,173.615,32.559,155.994
C02411=1064.759,282.819,405.470,173.616,32.563,155.995
C02412=1064.765,283.068,405.439,173.619,32.568,155.996
C02413=1064.771,283.315,405.409,173.622,32.571,155.996
C02414=1064.777,283.563,405.378,173.625,32.576,155.997
C02415=1064.783,283.811,405.347,173.628,32.579,155.998
C02416=1064.789,284.059,405.317,173.631,32.584,155.999
C02417=1064.796,284.307,405.286,173.633,32.588,155.999
C02418=1064.801,284.555,405.256,173.636,32.592,156.000
C02419=1064.807,284.803,405.225,173.639,32.596,156.001
C02420=1064.814,285.052,405.195,173.642,32.600,156.002
C02421=1064.819,285.299,405.164,173.645,32.604,156.002
C02422=1064.826,285.547,405.133,173.648,32.608,156.003
C02423=1064.832,285.795,405.102,173.650,32.612,156.004
C02424=1064.838,286.044,405.072,173.653,32.616,156.005
C02425=1064.844,286.292,405.041,173.656,32.620,156.005
C02426=1064.851,286.539,405.010,173.659,32.624,156.006
C02427=1064.857,286.787,404.980,173.662,32.628,156.007
C02428=1064.863,287.036,404.949,173.665,32.632,156.008
C02429=1064.869,287.284,404.919,173.668,32.636,156.008
C02430=1064.876,287.531,404.887,173.670,32.640,156.009
C02431=1064.882,287.779,404.857,173.672,32.645,156.010
C02432=1064.888,288.028,404.826,173.675,32.648,156.011
C02433=1064.894,288.275,404.795,173.678,32.653,156.012
C02434=1064.901,288.524,404.764,173.681,32.657,156.012
C02435=1064.906,288.771,404.734,173.684,32.661,156.013
C02436=1064.913,289.019,404.702,173.687,32.665,156.014
C02437=1064.918,289.267,404.672,173.690,32.669,156.015
C02438=1064.925,289.515,404.640,173.693,32.673,156.015
C02439=1064.931,289.742,404.612,173.695,32.677,156.016
C02440=1064.936,289.967,404.584,173.698,32.681,156.017
C02441=1064.942,290.194,404.556,173.701,32.684,156.018
C02442=1064.948,290.420,404.527,173.703,32.688,156.018
C02443=1064.953,290.646,404.499,173.706,32.692,156.019
C02444=1064.959,290.872,404.471,173.709,32.696,156.020
C02445=1064.965,291.099,404.443,173.711,32.699,156.020
C02446=1064.970,291.325,404.414,173.714,32.703,156.021
C02447=1064.976,291.572,404.383,173.717,32.707,156.022
C02448=1064.982,291.821,404.352,173.720,32.711,156.023
C02449=1064.988,292.068,404.321,173.723,32.715,156.023
C02450=1064.994,292.316,404.289,173.726,32.720,156.024
C02451=1065.001,292.565,404.258,173.729,32.724,156.025
C02452=1065.007,292.812,404.227,173.731,32.728,156.026
C02453=1065.013,293.061,404.196,173.734,32.732,156.027
C02454=1065.019,293.308,404.165,173.737,32.736,156.027
C02455=1065.025,293.556,404.133,173.740,32.740,156.028
C02456=1065.032,293.804,404.102,173.743,32.744,156.029
C02457=1065.037,294.052,404.071,173.745,32.749,156.030
C02458=1065.044,294.300,404.040,173.748,32.752,156.030
C02459=1065.051,294.548,404.008,173.751,32.757,156.031
C02460=1065.056,294.796,403.977,173.754,32.761,156.032
C02461=1065.062,295.044,403.946,173.757,32.765,156.033
C02462=1065.068,295.292,403.914,173.760,32.769,156.034
C02463=1065.075,295.539,403.883,173.763,32.773,156.034
C02464=1065.081,295.787,403.851,173.766,32.777,156.035
C02465=1065.087,296.035,403.819,173.769,32.782,156.036
C02466=1065.093,296.283,403.789,173.772,32.786,156.037
C02467=1065.099,296.531,403.757,173.775,32.790,156.038
C02468=1065.106,296.779,403.725,173.778,32.794,156.038
C02469=1065.111,297.027,403.694,173.781,32.799,156.039
C02470=1065.118,297.275,403.662,173.784,32.803,156.040
C02471=1065.124,297.523,403.630,173.787,32.807,156.041
C02472=1065.130,297.770,403.599,173.790,32.811,156.042
C02473=1065.136,298.018,403.567,173.793,32.815,156.042
C02474=1065.142,298.267,403.535,173.796,32.820,156.043
C02475=1065.147,298.514,403.503,173.799,32.824,156.044
C02476=1065.154,298.762,403.472,173.802,32.828,156.045
C02477=1065.160,299.010,403.440,173.805,32.832,156.046
C02478=1065.165,299.258,403.408,173.808,32.837,156.046
C02479=1065.172,299.506,403.377,173.811,32.841,156.047
C02480=1065.178,299.754,403.345,173.814,32.845,156.048
C02481=1065.184,300.001,403.312,173.817,32.849,156.049
C02482=1065.190,300.249,403.280,173.820,32.854,156.050
C02483=1065.197,300.497,403.249,173.823,32.858,156.051
C02484=1065.203,300.745,403.217,173.826,32.862,156.051
C02485=1065.208,300.993,403.185,173.829,32.866,156.052
C02486=1065.214,301.241,403.153,173.832,32.871,156.053
C02487=1065.221,301.488,403.121,173.835,32.875,156.054
C02488=1065.227,301.736,403.089,173.838,32.880,156.055
C02489=1065.233,301.985,403.057,173.841,32.884,156.056
C02490=1065.238,302.232,403.025,173.844,32.888,156.056
C02491=1065.245,302.479,402.993,173.847,32.892,156.057
C02492=1065.251,302.728,402.961,173.850,32.896,156.058
C02493=1065.257,302.976,402.929,173.853,32.901,156.059
C02494=1065.264,303.223,402.896,173.856,32.905,156.060
C02495=1065.269,303.457,402.867,173.859,32.909,156.060
C02496=1065.275,303.690,402.837,173.862,32.913,156.061
C02497=1065.281,303.924,402.807,173.865,32.917,156.062
C02498=1065.286,304.158,402.776,173.867,32.921,156.063
C02499=1065.293,304.391,402.746,173.870,32.925,156.064
C02500=1065.298,304.625,402.715,173.873,32.929,156.064
C02501=1065.304,304.859,402.685,173.876,32.933,156.065
C02502=1065.310,305.093,402.655,173.879,32.937,156.066
C02503=1065.316,305.341,402.622,173.882,32.942,156.067
C02504=1065.323,305.588,402.591,173.885,32.946,156.068
C02505=1065.329,305.836,402.558,173.888,32.950,156.068
C02506=1065.335,306.084,402.526,173.891,32.954,156.069
C02507=1065.341,306.332,402.493,173.894,32.959,156.070
C02508=1065.347,306.580,402.461,173.897,32.963,156.071
C02509=1065.354,306.827,402.429,173.901,32.968,156.072
C02510=1065.360,307.076,402.397,173.904,32.972,156.073
C02511=1065.366,307.322,402.364,173.907,32.976,156.073
C02512=1065.372,307.571,402.332,173.910,32.980,156.074
C02513=1065.378,307.818,402.300,173.913,32.985,156.075
C02514=1065.385,308.066,402.267,173.916,32.989,156.076
C02515=1065.391,308.314,402.235,173.919,32.993,156.077
C02516=1065.398,308.561,402.203,173.922,32.998,156.078
C02517=1065.404,308.809,402.170,173.925,33.002,156.078
C02518=1065.411,309.058,402.138,173.929,33.006,156.079
C02519=1065.417,309.305,402.105,173.932,33.010,156.080
C02520=1065.423,309.553,402.072,173.935,33.015,156.081
C02521=1065.429,309.801,402.040,173.938,33.019,156.082
C02522=1065.435,310.049,402.007,173.941,33.024,156.083
C02523=1065.442,310.296,401.975,173.944,33.028,156.083
C02524=1065.449,310.544,401.943,173.947,33.032,156.084
C02525=1065.455,310.791,401.910,173.951,33.036,156.085
C02526=1065.461,311.039,401.878,173.954,33.041,156.086
C02527=1065.467,311.287,401.845,173.957,33.045,156.087
C02528=1065.474,311.535,401.812,173.960,33.049,156.088
C02529=1065.480,311.782,401.780,173.963,33.054,156.088
C02530=1065.487,312.031,401.746,173.966,33.058,156.089
C02531=1065.493,312.278,401.714,173.970,33.062,156.090
C02532=1065.499,312.526,401.682,173.973,33.067,156.091
C02533=1065.505,312.774,401.649,173.976,33.071,156.092
C02534=1065.512,313.022,401.616,173.979,33.075,156.093
C02535=1065.519,313.269,401.584,173.982,33.080,156.093
C02536=1065.526,313.517,401.551,173.985,33.084,156.094
C02537=1065.532,313.765,401.518,173.989,33.089,156.095
C02538=1065.538,314.012,401.485,173.992,33.093,156.096
C02539=1065.544,314.260,401.452,173.995,33.098,156.097
C02540=1065.550,314.508,401.419,173.998,33.102,156.098
C02541=1065.556,314.755,401.387,174.001,33.106,156.099
C02542=1065.562,315.003,401.353,174.004,33.111,156.099
C02543=1065.568,315.250,401.320,174.008,33.116,156.100
C02544=1065.575,315.499,401.286,174.011,33.120,156.101
C02545=1065.581,315.746,401.253,174.014,33.124,156.102
C02546=1065.586,315.994,401.220,174.017,33.129,156.103
C02547=1065.593,316.242,401.187,174.020,33.133,156.104
C02548=1065.599,316.489,401.154,174.023,33.138,156.105
C02549=1065.605,316.737,401.120,174.027,33.142,156.106
C02550=1065.612,316.985,401.087,174.031,33.147,156.107
C02551=1065.618,317.224,401.055,174.034,33.151,156.107
C02552=1065.623,317.463,401.022,174.037,33.156,156.108
C02553=1065.629,317.702,400.991,174.040,33.160,156.109
C02554=1065.635,317.942,400.959,174.043,33.164,156.110
C02555=1065.641,318.180,400.927,174.046,33.169,156.111
C02556=1065.648,318.419,400.895,174.049,33.173,156.112
C02557=1065.653,318.658,400.862,174.053,33.178,156.113
C02558=1065.659,318.897,400.830,174.056,33.182,156.114
C02559=1065.665,319.141,400.797,174.059,33.187,156.114
C02560=1065.672,319.386,400.764,174.062,33.191,156.115
C02561=1065.677,319.630,400.732,174.065,33.195,156.116
C02562=1065.683,319.874,400.698,174.068,33.200,156.117
C02563=1065.689,320.118,400.665,174.072,33.205,156.118
C02564=1065.696,320.363,400.632,174.075,33.209,156.119
C02565=1065.702,320.607,400.599,174.078,33.214,156.120
C02566=1065.708,320.850,400.566,174.081,33.218,156.121
C02567=1065.714,321.098,400.533,174.084,33.223,156.122
C02568=1065.721,321.346,400.499,174.088,33.228,156.123
C02569=1065.727,321.593,400.465,174.091,33.232,156.123
C02570=1065.733,321.841,400.432,174.094,33.237,156.124
C02571=1065.740,322.089,400.398,174.097,33.241,156.125
C02572=1065.746,322.336,400.365,174.101,33.246,156.126
C02573=1065.752,322.584,400.331,174.105,33.250,156.127
C02574=1065.759,322.832,400.298,174.108,33.255,156.128
C02575=1065.765,323.079,400.264,174.111,33.260,156.129
C02576=1065.772,323.327,400.230,174.115,33.264,156.130
C02577=1065.777,323.575,400.197,174.118,33.269,156.131
C02578=1065.785,323.823,400.163,174.121,33.273,156.132
C02579=1065.790,324.070,400.129,174.125,33.278,156.133
C02580=1065.797,324.318,400.095,174.128,33.282,156.133
C02581=1065.803,324.565,400.062,174.131,33.287,156.134
C02582=1065.809,324.813,400.028,174.135,33.292,156.135
C02583=1065.816,325.060,399.994,174.138,33.297,156.136
C02584=1065.822,325.308,399.960,174.141,33.301,156.137
C02585=1065.829,325.556,399.927,174.144,33.306,156.138
C02586=1065.835,325.803,399.893,174.148,33.310,156.139
C02587=1065.841,326.051,399.858,174.151,33.315,156.140
C02588=1065.848,326.299,399.824,174.154,33.320,156.141
C02589=1065.854,326.546,399.790,174.158,33.325,156.142
C02590=1065.862,326.794,399.757,174.162,33.329,156.143
C02591=1065.867,327.041,399.723,174.165,33.333,156.144
C02592=1065.874,327.289,399.688,174.169,33.338,156.144
C02593=1065.880,327.537,399.655,174.172,33.343,156.145
C02594=1065.887,327.785,399.621,174.176,33.348,156.146
C02595=1065.893,328.033,399.587,174.179,33.352,156.147
C02596=1065.900,328.280,399.553,174.182,33.357,156.148
C02597=1065.906,328.528,399.519,174.186,33.362,156.149
C02598=1065.913,328.775,399.485,174.189,33.367,156.150
C02599=1065.919,329.023,399.451,174.192,33.371,156.151
C02600=1065.926,329.271,399.416,174.196,33.376,156.152
C02601=1065.933,329.517,399.382,174.199,33.380,156.153
C02602=1065.939,329.765,399.348,174.203,33.385,156.154
C02603=1065.945,330.013,399.313,174.207,33.390,156.155
C02604=1065.952,330.260,399.280,174.210,33.395,156.156
C02605=1065.959,330.508,399.245,174.214,33.399,156.157
C02606=1065.965,330.756,399.211,174.217,33.404,156.158
C02607=1065.971,330.988,399.179,174.220,33.409,156.159
C02608=1065.977,331.221,399.147,174.223,33.413,156.159
C02609=1065.984,331.454,399.115,174.227,33.418,156.160
C02610=1065.989,331.686,399.082,174.230,33.422,156.161
C02611=1065.995,331.919,399.050,174.233,33.426,156.162
C02612=1066.001,332.151,399.017,174.236,33.431,156.163
C02613=1066.007,332.384,398.984,174.239,33.436,156.164
C02614=1066.013,332.616,398.952,174.243,33.441,156.165
C02615=1066.019,332.863,398.918,174.247,33.445,156.166
C02616=1066.026,333.111,398.883,174.250,33.450,156.167
C02617=1066.032,333.359,398.848,174.254,33.455,156.168
C02618=1066.038,333.606,398.814,174.257,33.460,156.169
C02619=1066.045,333.853,398.779,174.261,33.465,156.170
C02620=1066.051,334.101,398.745,174.264,33.470,156.171
C02621=1066.058,334.348,398.710,174.268,33.475,156.172
C02622=1066.064,334.596,398.675,174.271,33.480,156.173
C02623=1066.070,334.844,398.641,174.274,33.484,156.174
C02624=1066.077,335.091,398.606,174.278,33.490,156.175
C02625=1066.084,335.339,398.571,174.282,33.494,156.176
C02626=1066.090,335.586,398.537,174.286,33.499,156.177
C02627=1066.097,335.833,398.501,174.289,33.504,156.178
C02628=1066.102,336.082,398.466,174.293,33.509,156.179
C02629=1066.109,336.329,398.431,174.296,33.514,156.180
C02630=1066.115,336.576,398.397,174.300,33.519,156.181
C02631=1066.122,336.824,398.362,174.303,33.524,156.182
C02632=1066.129,337.071,398.327,174.307,33.528,156.183
C02633=1066.135,337.319,398.293,174.310,33.534,156.184
C02634=1066.142,337.566,398.257,174.315,33.538,156.185
C02635=1066.149,337.814,398.222,174.318,33.544,156.186
C02636=1066.154,338.061,398.187,174.321,33.549,156.187
C02637=1066.160,338.309,398.153,174.325,33.554,156.188
C02638=1066.167,338.556,398.117,174.328,33.559,156.189
C02639=1066.173,338.804,398.082,174.332,33.564,156.190
C02640=1066.180,339.051,398.047,174.335,33.569,156.191
C02641=1066.187,339.299,398.011,174.339,33.574,156.192
C02642=1066.194,339.546,397.976,174.343,33.579,156.193
C02643=1066.199,339.794,397.942,174.347,33.584,156.194
C02644=1066.205,340.041,397.907,174.350,33.589,156.195
C02645=1066.212,340.288,397.871,174.354,33.594,156.196
C02646=1066.218,340.536,397.836,174.357,33.599,156.197
C02647=1066.225,340.783,397.801,174.361,33.604,156.198
C02648=1066.232,341.031,397.765,174.365,33.609,156.199
C02649=1066.238,341.278,397.730,174.368,33.615,156.200
C02650=1066.245,341.526,397.695,174.373,33.620,156.201
C02651=1066.251,341.773,397.659,174.376,33.624,156.202
C02652=1066.257,342.021,397.624,174.380,33.630,156.203
C02653=1066.264,342.268,397.589,174.383,33.635,156.205
C02654=1066.271,342.515,397.553,174.387,33.640,156.205
C02655=1066.277,342.763,397.518,174.390,33.645,156.207
C02656=1066.284,343.011,397.483,174.394,33.650,156.208
C02657=1066.291,343.257,397.447,174.398,33.655,156.209
C02658=1066.297,343.505,397.411,174.402,33.661,156.210
C02659=1066.304,343.752,397.376,174.406,33.665,156.211
C02660=1066.310,344.000,397.340,174.409,33.671,156.212
C02661=1066.316,344.247,397.305,174.413,33.676,156.213
C02662=1066.323,344.494,397.268,174.416,33.681,156.214
C02663=1066.328,344.724,397.236,174.420,33.686,156.215
C02664=1066.334,344.955,397.202,174.424,33.691,156.216
C02665=1066.341,345.185,397.169,174.427,33.696,156.217
C02666=1066.346,345.415,397.136,174.431,33.701,156.218
C02667=1066.353,345.645,397.102,174.434,33.706,156.219
C02668=1066.359,345.876,397.069,174.437,33.711,156.220
C02669=1066.364,346.106,397.036,174.441,33.716,156.221
C02670=1066.371,346.336,397.003,174.444,33.720,156.222
C02671=1066.378,346.583,396.967,174.449,33.725,156.223
C02672=1066.384,346.831,396.931,174.452,33.731,156.224
C02673=1066.391,347.077,396.896,174.456,33.736,156.225
C02674=1066.397,347.325,396.860,174.460,33.742,156.227
C02675=1066.403,347.572,396.823,174.463,33.747,156.228
C02676=1066.410,347.819,396.788,174.467,33.752,156.229
C02677=1066.417,348.067,396.751,174.471,33.757,156.230
C02678=1066.423,348.315,396.716,174.475,33.763,156.231
C02679=1066.430,348.562,396.680,174.479,33.768,156.232
C02680=1066.436,348.809,396.643,174.482,33.774,156.233
C02681=1066.442,349.056,396.608,174.486,33.779,156.234
C02682=1066.449,349.303,396.572,174.490,33.784,156.235
C02683=1066.456,349.551,396.535,174.494,33.790,156.237
C02684=1066.462,349.799,396.499,174.498,33.795,156.238
C02685=1066.469,350.046,396.463,174.502,33.800,156.239
C02686=1066.476,350.292,396.427,174.505,33.806,156.240
C02687=1066.482,350.540,396.391,174.509,33.811,156.241
C02688=1066.489,350.788,396.354,174.514,33.817,156.242
C02689=1066.496,351.035,396.319,174.517,33.822,156.243
C02690=1066.502,351.282,396.282,174.521,33.828,156.244
C02691=1066.508,351.529,396.246,174.525,33.833,156.246
C02692=1066.515,351.777,396.210,174.528,33.839,156.247
C02693=1066.522,352.024,396.173,174.533,33.844,156.248
C02694=1066.529,352.271,396.137,174.537,33.850,156.249
C02695=1066.535,352.518,396.101,174.541,33.855,156.250
C02696=1066.542,352.766,396.064,174.544,33.861,156.251
C02697=1066.548,353.013,396.028,174.548,33.866,156.252
C02698=1066.555,353.260,395.991,174.553,33.872,156.254
C02699=1066.561,353.507,395.954,174.556,33.877,156.255
C02700=1066.568,353.755,395.918,174.560,33.883,156.256
C02701=1066.574,354.002,395.881,174.564,33.888,156.257
C02702=1066.581,354.249,395.845,174.568,33.894,156.258
C02703=1066.587,354.496,395.808,174.572,33.899,156.259
C02704=1066.594,354.743,395.772,174.576,33.905,156.261
C02705=1066.601,354.991,395.735,174.580,33.910,156.262
C02706=1066.607,355.238,395.699,174.584,33.916,156.263
C02707=1066.614,355.485,395.661,174.587,33.922,156.264
C02708=1066.621,355.732,395.625,174.592,33.927,156.265
C02709=1066.627,355.979,395.588,174.596,33.933,156.267
C02710=1066.633,356.227,395.552,174.600,33.939,156.268
C02711=1066.640,356.474,395.515,174.603,33.944,156.269
C02712=1066.647,356.721,395.478,174.608,33.950,156.270
C02713=1066.654,356.969,395.441,174.612,33.955,156.271
C02714=1066.660,357.216,395.404,174.616,33.961,156.272
C02715=1066.667,357.463,395.367,174.619,33.967,156.274
C02716=1066.674,357.710,395.330,174.623,33.972,156.275
C02717=1066.681,357.958,395.294,174.628,33.978,156.276
C02718=1066.687,358.204,395.256,174.632,33.984,156.277
C02719=1066.694,358.436,395.222,174.635,33.989,156.278
C02720=1066.700,358.668,395.188,174.639,33.994,156.280
C02721=1066.706,358.900,395.153,174.644,34.000,156.281
C02722=1066.713,359.133,395.118,174.647,34.005,156.282
C02723=1066.719,359.364,395.083,174.651,34.011,156.283
C02724=1066.725,359.596,395.048,174.654,34.016,156.284
C02725=1066.731,359.829,395.013,174.659,34.022,156.285
C02726=1066.737,360.061,394.978,174.663,34.027,156.286
C02727=1066.744,360.308,394.941,174.666,34.033,156.288
C02728=1066.751,360.555,394.904,174.670,34.039,156.289
C02729=1066.758,360.802,394.867,174.675,34.045,156.290
C02730=1066.764,361.049,394.829,174.679,34.051,156.292
C02731=1066.771,361.297,394.792,174.683,34.056,156.293
C02732=1066.778,361.544,394.755,174.687,34.062,156.294
C02733=1066.785,361.791,394.717,174.691,34.068,156.295
C02734=1066.791,362.038,394.681,174.695,34.074,156.297
C02735=1066.798,362.285,394.643,174.699,34.080,156.298
C02736=1066.805,362.532,394.605,174.703,34.085,156.299
C02737=1066.812,362.779,394.568,174.708,34.092,156.300
C02738=1066.818,363.026,394.530,174.712,34.097,156.302
C02739=1066.825,363.273,394.493,174.716,34.104,156.303
C02740=1066.832,363.520,394.456,174.720,34.110,156.304
C02741=1066.839,363.768,394.419,174.724,34.115,156.305
C02742=1066.845,364.014,394.381,174.728,34.121,156.307
C02743=1066.852,364.261,394.343,174.732,34.127,156.308
C02744=1066.859,364.509,394.306,174.737,34.133,156.309
C02745=1066.865,364.755,394.268,174.741,34.139,156.310
C02746=1066.872,365.002,394.230,174.745,34.145,156.312
C02747=1066.879,365.250,394.192,174.749,34.152,156.313
C02748=1066.886,365.496,394.155,174.754,34.157,156.314
C02749=1066.892,365.744,394.117,174.758,34.164,156.316
C02750=1066.899,365.991,394.079,174.762,34.170,156.317
C02751=1066.906,366.237,394.041,174.767,34.176,156.318
C02752=1066.912,366.484,394.003,174.770,34.182,156.320
C02753=1066.919,366.732,393.965,174.774,34.188,156.321
C02754=1066.926,366.979,393.927,174.779,34.194,156.322
C02755=1066.932,367.225,393.890,174.783,34.201,156.324
C02756=1066.939,367.472,393.851,174.787,34.207,156.325
C02757=1066.947,367.719,393.814,174.792,34.213,156.326
C02758=1066.953,367.967,393.776,174.796,34.219,156.328
C02759=1066.959,368.214,393.738,174.800,34.225,156.329
C02760=1066.967,368.460,393.700,174.804,34.231,156.330
C02761=1066.973,368.708,393.662,174.809,34.238,156.332
C02762=1066.980,368.955,393.624,174.813,34.244,156.333
C02763=1066.987,369.202,393.585,174.817,34.250,156.334
C02764=1066.994,369.449,393.548,174.822,34.256,156.336
C02765=1067.001,369.695,393.509,174.826,34.263,156.337
C02766=1067.007,369.942,393.471,174.830,34.269,156.339
C02767=1067.015,370.189,393.433,174.835,34.275,156.340
C02768=1067.021,370.436,393.395,174.839,34.281,156.341
C02769=1067.028,370.683,393.356,174.843,34.288,156.343
C02770=1067.035,370.930,393.318,174.848,34.294,156.344
C02771=1067.042,371.177,393.279,174.852,34.301,156.345
C02772=1067.049,371.424,393.242,174.857,34.307,156.347
C02773=1067.056,371.671,393.203,174.861,34.313,156.348
C02774=1067.063,371.918,393.164,174.865,34.319,156.350
C02775=1067.069,372.159,393.128,174.870,34.326,156.351
C02776=1067.076,372.399,393.090,174.874,34.332,156.352
C02777=1067.083,372.640,393.052,174.878,34.338,156.354
C02778=1067.090,372.880,393.015,174.883,34.344,156.355
C02779=1067.097,373.121,392.978,174.887,34.350,156.356
C02780=1067.103,373.362,392.939,174.891,34.357,156.358
C02781=1067.110,373.603,392.902,174.896,34.363,156.359
C02782=1067.117,373.844,392.864,174.900,34.370,156.361
C02783=1067.123,374.091,392.826,174.904,34.376,156.362
C02784=1067.130,374.338,392.787,174.909,34.383,156.363
C02785=1067.137,374.585,392.748,174.913,34.389,156.365
C02786=1067.143,374.831,392.709,174.918,34.396,156.366
C02787=1067.150,375.078,392.670,174.922,34.402,156.368
C02788=1067.157,375.325,392.632,174.926,34.409,156.369
C02789=1067.164,375.572,392.593,174.932,34.416,156.371
C02790=1067.171,375.819,392.554,174.936,34.422,156.372
C02791=1067.178,376.065,392.516,174.941,34.429,156.374
C02792=1067.185,376.312,392.477,174.945,34.436,156.375
C02793=1067.192,376.558,392.437,174.949,34.442,156.377
C02794=1067.199,376.805,392.398,174.954,34.449,156.378
C02795=1067.206,377.052,392.360,174.958,34.455,156.379
C02796=1067.213,377.299,392.320,174.963,34.462,156.381
C02797=1067.220,377.546,392.282,174.968,34.469,156.382
C02798=1067.227,377.793,392.243,174.972,34.476,156.384
C02799=1067.234,378.039,392.203,174.977,34.482,156.385
C02800=1067.241,378.286,392.164,174.981,34.489,156.387
C02801=1067.248,378.533,392.126,174.986,34.496,156.388
C02802=1067.255,378.780,392.086,174.990,34.502,156.390
C02803=1067.262,379.027,392.047,174.996,34.509,156.391
C02804=1067.269,379.274,392.008,175.000,34.516,156.393
C02805=1067.276,379.520,391.968,175.004,34.523,156.394
C02806=1067.283,379.767,391.930,175.009,34.530,156.396
C02807=1067.291,380.013,391.890,175.013,34.537,156.398
C02808=1067.297,380.260,391.851,175.019,34.543,156.399
C02809=1067.305,380.506,391.811,175.023,34.550,156.401
C02810=1067.311,380.754,391.771,175.028,34.557,156.402
C02811=1067.318,381.001,391.732,175.032,34.564,156.404
C02812=1067.325,381.247,391.693,175.037,34.571,156.405
C02813=1067.332,381.494,391.653,175.042,34.578,156.407
C02814=1067.340,381.741,391.614,175.047,34.585,156.408
C02815=1067.346,381.988,391.574,175.051,34.592,156.410
C02816=1067.353,382.234,391.535,175.055,34.599,156.411
C02817=1067.360,382.481,391.496,175.061,34.606,156.413
C02818=1067.367,382.728,391.455,175.065,34.613,156.415
C02819=1067.374,382.974,391.416,175.070,34.620,156.416
C02820=1067.381,383.220,391.376,175.074,34.627,156.418
C02821=1067.388,383.467,391.336,175.080,34.634,156.419
C02822=1067.395,383.714,391.297,175.084,34.641,156.421
C02823=1067.402,383.960,391.257,175.089,34.648,156.423
C02824=1067.409,384.208,391.217,175.093,34.656,156.424
C02825=1067.416,384.454,391.177,175.099,34.663,156.426
C02826=1067.424,384.701,391.137,175.103,34.670,156.427
C02827=1067.430,384.947,391.097,175.108,34.677,156.429
C02828=1067.437,385.194,391.058,175.113,34.684,156.431
C02829=1067.445,385.440,391.018,175.118,34.691,156.432
C02830=1067.452,385.687,390.977,175.122,34.699,156.434
C02831=1067.460,385.952,390.935,175.128,34.706,156.436
C02832=1067.467,386.217,390.891,175.134,34.714,156.437
C02833=1067.475,386.482,390.848,175.138,34.722,156.439
C02834=1067.483,386.746,390.805,175.144,34.730,156.441
C02835=1067.490,386.994,390.765,175.148,34.738,156.443
C02836=1067.497,387.240,390.725,175.154,34.745,156.444
C02837=1067.505,387.487,390.685,175.158,34.752,156.446
C02838=1067.511,387.733,390.644,175.163,34.759,156.448
C02839=1067.519,387.980,390.604,175.168,34.766,156.449
C02840=1067.525,388.226,390.564,175.173,34.774,156.451
C02841=1067.533,388.472,390.524,175.179,34.781,156.453
C02842=1067.540,388.720,390.483,175.183,34.789,156.454
C02843=1067.547,388.966,390.444,175.188,34.796,156.456
C02844=1067.555,389.212,390.402,175.193,34.804,156.458
C02845=1067.562,389.459,390.363,175.198,34.811,156.459
C02846=1067.569,389.705,390.322,175.203,34.819,156.461
C02847=1067.577,389.952,390.282,175.208,34.826,156.463
C02848=1067.584,390.198,390.241,175.213,34.834,156.464
C02849=1067.591,390.445,390.201,175.218,34.841,156.466
C02850=1067.599,390.691,390.160,175.223,34.848,156.468
C02851=1067.606,390.938,390.120,175.228,34.856,156.470
C02852=1067.613,391.184,390.079,175.233,34.864,156.471
C02853=1067.621,391.431,390.038,175.239,34.872,156.473
C02854=1067.628,391.678,389.998,175.243,34.879,156.475
C02855=1067.635,391.924,389.957,175.249,34.887,156.477
C02856=1067.642,392.170,389.916,175.253,34.894,156.478
C02857=1067.650,392.417,389.875,175.259,34.902,156.480
C02858=1067.656,392.663,389.835,175.264,34.910,156.482
C02859=1067.664,392.910,389.794,175.269,34.918,156.484
C02860=1067.672,393.156,389.753,175.274,34.926,156.486
C02861=1067.679,393.403,389.712,175.280,34.934,156.487
C02862=1067.686,393.649,389.670,175.284,34.941,156.489
C02863=1067.693,393.895,389.630,175.290,34.949,156.491
C02864=1067.700,394.142,389.588,175.294,34.957,156.493
C02865=1067.708,394.388,389.547,175.300,34.965,156.495
C02866=1067.716,394.635,389.507,175.305,34.973,156.496
C02867=1067.723,394.881,389.465,175.310,34.980,156.498
C02868=1067.730,395.128,389.424,175.315,34.989,156.500
C02869=1067.737,395.374,389.383,175.321,34.996,156.502
C02870=1067.744,395.620,389.342,175.325,35.004,156.504
C02871=1067.751,395.867,389.301,175.331,35.012,156.506
C02872=1067.759,396.113,389.260,175.337,35.020,156.507
C02873=1067.766,396.359,389.218,175.342,35.029,156.509
C02874=1067.774,396.606,389.176,175.347,35.036,156.511
C02875=1067.781,396.853,389.135,175.352,35.045,156.513
C02876=1067.788,397.099,389.094,175.358,35.053,156.515
C02877=1067.796,397.345,389.052,175.362,35.061,156.517
C02878=1067.803,397.592,389.011,175.368,35.069,156.519
C02879=1067.811,397.838,388.970,175.374,35.077,156.521
C02880=1067.818,398.084,388.928,175.378,35.085,156.522
C02881=1067.825,398.331,388.886,175.384,35.093,156.524
C02882=1067.833,398.577,388.844,175.390,35.102,156.526
C02883=1067.840,398.823,388.803,175.395,35.110,156.528
C02884=1067.848,399.069,388.761,175.400,35.118,156.530
C02885=1067.855,399.316,388.720,175.405,35.126,156.532
C02886=1067.863,399.563,388.678,175.411,35.135,156.534
C02887=1067.871,399.844,388.630,175.417,35.144,156.536
C02888=1067.879,400.125,388.583,175.424,35.154,156.538
C02889=1067.888,400.405,388.535,175.430,35.163,156.541
C02890=1067.896,400.687,388.487,175.435,35.173,156.543
C02891=1067.904,400.933,388.445,175.441,35.181,156.545
C02892=1067.911,401.179,388.403,175.447,35.190,156.547
C02893=1067.920,401.426,388.361,175.453,35.198,156.549
C02894=1067.927,401.672,388.320,175.458,35.207,156.551
C02895=1067.934,401.919,388.277,175.463,35.215,156.553
C02896=1067.941,402.165,388.235,175.469,35.224,156.555
C02897=1067.949,402.411,388.193,175.475,35.232,156.557
C02898=1067.957,402.657,388.151,175.480,35.241,156.559
C02899=1067.964,402.904,388.108,175.486,35.250,156.561
C02900=1067.972,403.150,388.066,175.492,35.258,156.563
C02901=1067.980,403.396,388.024,175.497,35.266,156.565
C02902=1067.987,403.642,387.982,175.502,35.275,156.567
C02903=1067.995,403.889,387.939,175.508,35.284,156.569
C02904=1068.002,404.135,387.897,175.514,35.293,156.571
C02905=1068.009,404.381,387.855,175.520,35.302,156.573
C02906=1068.017,404.628,387.812,175.526,35.310,156.575
C02907=1068.025,404.874,387.769,175.530,35.319,156.577
C02908=1068.032,405.120,387.727,175.536,35.328,156.580
C02909=1068.040,405.366,387.685,175.542,35.337,156.582
C02910=1068.047,405.613,387.642,175.548,35.346,156.584
C02911=1068.056,405.859,387.599,175.554,35.354,156.586
C02912=1068.063,406.105,387.557,175.560,35.364,156.588
C02913=1068.071,406.352,387.514,175.566,35.372,156.590
C02914=1068.078,406.597,387.471,175.571,35.381,156.592
C02915=1068.085,406.844,387.428,175.577,35.390,156.594
C02916=1068.093,407.090,387.386,175.583,35.399,156.597
C02917=1068.101,407.337,387.343,175.589,35.409,156.599
C02918=1068.109,407.582,387.300,175.594,35.418,156.601
C02919=1068.116,407.829,387.257,175.600,35.427,156.603
C02920=1068.123,408.075,387.214,175.606,35.436,156.605
C02921=1068.132,408.321,387.171,175.612,35.445,156.607
C02922=1068.139,408.567,387.128,175.618,35.454,156.610
C02923=1068.146,408.813,387.085,175.624,35.463,156.612
C02924=1068.154,409.059,387.042,175.630,35.472,156.614
C02925=1068.162,409.306,386.999,175.636,35.482,156.616
C02926=1068.170,409.552,386.956,175.642,35.491,156.619
C02927=1068.177,409.797,386.913,175.648,35.500,156.621
C02928=1068.185,410.044,386.869,175.654,35.510,156.623
C02929=1068.193,410.290,386.826,175.660,35.519,156.625
C02930=1068.200,410.536,386.782,175.666,35.528,156.627
C02931=1068.209,410.782,386.739,175.672,35.538,156.630
C02932=1068.216,411.028,386.696,175.678,35.547,156.632
C02933=1068.224,411.275,386.652,175.684,35.556,156.634
C02934=1068.232,411.520,386.609,175.690,35.566,156.637
C02935=1068.240,411.766,386.566,175.696,35.576,156.639
C02936=1068.248,412.013,386.522,175.702,35.585,156.641
C02937=1068.255,412.259,386.479,175.709,35.595,156.643
C02938=1068.264,412.505,386.436,175.715,35.604,156.646
C02939=1068.271,412.751,386.392,175.721,35.614,156.648
C02940=1068.279,412.997,386.348,175.728,35.623,156.650
C02941=1068.287,413.243,386.304,175.734,35.633,156.653
C02942=1068.295,413.489,386.261,175.740,35.642,156.655
C02943=1068.304,413.774,386.210,175.747,35.654,156.658
C02944=1068.313,414.059,386.160,175.754,35.665,156.661
C02945=1068.322,414.344,386.108,175.762,35.676,156.663
C02946=1068.332,414.629,386.058,175.769,35.687,156.666
C02947=1068.340,414.876,386.015,175.775,35.698,156.668
C02948=1068.348,415.121,385.970,175.781,35.707,156.671
C02949=1068.356,415.367,385.926,175.789,35.717,156.673
C02950=1068.363,415.614,385.882,175.795,35.727,156.676
C02951=1068.372,415.859,385.838,175.801,35.737,156.678
C02952=1068.379,416.106,385.794,175.807,35.747,156.681
C02953=1068.387,416.351,385.750,175.814,35.758,156.683
C02954=1068.395,416.597,385.706,175.820,35.767,156.685
C02955=1068.403,416.843,385.661,175.827,35.777,156.688
C02956=1068.411,417.089,385.616,175.833,35.787,156.690
C02957=1068.419,417.335,385.573,175.840,35.798,156.693
C02958=1068.427,417.581,385.528,175.846,35.808,156.695
C02959=1068.435,417.827,385.484,175.853,35.818,156.698
C02960=1068.443,418.073,385.439,175.860,35.829,156.701
C02961=1068.451,418.319,385.395,175.866,35.839,156.703
C02962=1068.460,418.565,385.351,175.872,35.849,156.706
C02963=1068.468,418.810,385.306,175.880,35.859,156.708
C02964=1068.475,419.057,385.261,175.886,35.870,156.711
C02965=1068.484,419.303,385.217,175.893,35.880,156.713
C02966=1068.492,419.548,385.172,175.899,35.890,156.716
C02967=1068.500,419.794,385.127,175.906,35.900,156.718
C02968=1068.508,420.040,385.083,175.913,35.911,156.721
C02969=1068.517,420.286,385.038,175.919,35.922,156.724
C02970=1068.524,420.531,384.993,175.927,35.932,156.726
C02971=1068.532,420.777,384.948,175.933,35.942,156.729
C02972=1068.541,421.024,384.904,175.940,35.953,156.731
C02973=1068.550,421.269,384.859,175.947,35.964,156.734
C02974=1068.557,421.515,384.814,175.954,35.974,156.737
C02975=1068.566,421.761,384.768,175.961,35.985,156.739
C02976=1068.573,422.007,384.723,175.968,35.996,156.742
C02977=1068.582,422.252,384.678,175.974,36.007,156.745
C02978=1068.589,422.499,384.633,175.982,36.017,156.747
C02979=1068.598,422.744,384.588,175.988,36.028,156.750
C02980=1068.606,422.989,384.543,175.996,36.039,156.753
C02981=1068.614,423.236,384.497,176.002,36.050,156.755
C02982=1068.623,423.481,384.452,176.009,36.061,156.758
C02983=1068.631,423.727,384.406,176.017,36.072,156.761
C02984=1068.639,423.972,384.361,176.023,36.083,156.764
C02985=1068.647,424.218,384.315,176.031,36.094,156.766
C02986=1068.656,424.463,384.270,176.038,36.105,156.769
C02987=1068.664,424.709,384.224,176.045,36.116,156.772
C02988=1068.672,424.955,384.180,176.052,36.127,156.775
C02989=1068.680,425.201,384.134,176.060,36.138,156.778
C02990=1068.689,425.446,384.088,176.066,36.149,156.780
C02991=1068.697,425.692,384.042,176.074,36.160,156.783
C02992=1068.706,425.938,383.997,176.081,36.172,156.786
C02993=1068.714,426.183,383.951,176.088,36.183,156.789
C02994=1068.723,426.429,383.906,176.096,36.194,156.792
C02995=1068.731,426.675,383.860,176.103,36.206,156.795
C02996=1068.740,426.920,383.814,176.111,36.217,156.797
C02997=1068.748,427.166,383.768,176.117,36.228,156.800
C02998=1068.756,427.412,383.722,176.125,36.240,156.803
C02999=1068.767,427.716,383.665,176.134,36.254,156.807
C03000=1068.777,428.020,383.608,176.144,36.268,156.810
C03001=1068.788,428.324,383.550,176.153,36.283,156.814
C03002=1068.798,428.629,383.493,176.162,36.297,156.818
C03003=1068.807,428.875,383.447,176.170,36.309,156.821
C03004=1068.815,429.120,383.401,176.177,36.321,156.824
C03005=1068.824,429.366,383.354,176.185,36.332,156.827
C03006=1068.832,429.611,383.309,176.193,36.344,156.830
C03007=1068.841,429.856,383.262,176.201,36.356,156.833
C03008=1068.849,430.102,383.215,176.208,36.368,156.836
C03009=1068.858,430.347,383.169,176.215,36.379,156.839
C03010=1068.867,430.593,383.122,176.223,36.391,156.842
C03011=1068.875,430.838,383.076,176.231,36.403,156.845
C03012=1068.884,431.084,383.029,176.238,36.415,156.848
C03013=1068.893,431.329,382.982,176.246,36.427,156.851
C03014=1068.901,431.575,382.936,176.254,36.439,156.854
C03015=1068.910,431.820,382.889,176.262,36.451,156.857
C03016=1068.918,432.066,382.842,176.270,36.464,156.860
C03017=1068.927,432.311,382.795,176.278,36.476,156.863
C03018=1068.935,432.557,382.749,176.286,36.488,156.867
C03019=1068.944,432.802,382.701,176.294,36.500,156.870
C03020=1068.953,433.047,382.654,176.302,36.513,156.873
C03021=1068.961,433.293,382.608,176.310,36.525,156.876
C03022=1068.970,433.537,382.560,176.318,36.538,156.879
C03023=1068.979,433.783,382.514,176.326,36.550,156.883
C03024=1068.987,434.028,382.466,176.334,36.562,156.886
C03025=1068.995,434.274,382.419,176.342,36.575,156.889
C03026=1069.005,434.519,382.371,176.351,36.588,156.892
C03027=1069.014,434.764,382.324,176.359,36.600,156.896
C03028=1069.022,435.010,382.277,176.367,36.613,156.899
C03029=1069.031,435.255,382.229,176.375,36.626,156.902
C03030=1069.040,435.499,382.182,176.383,36.638,156.905
C03031=1069.049,435.746,382.135,176.392,36.651,156.909
C03032=1069.058,435.991,382.087,176.400,36.663,156.912
C03033=1069.066,436.236,382.039,176.408,36.676,156.915
C03034=1069.075,436.481,381.992,176.417,36.689,156.919
C03035=1069.084,436.726,381.944,176.425,36.702,156.922
C03036=1069.093,436.971,381.897,176.433,36.715,156.926
C03037=1069.103,437.217,381.849,176.442,36.728,156.929
C03038=1069.111,437.462,381.801,176.451,36.741,156.932
C03039=1069.121,437.707,381.754,176.459,36.754,156.936
C03040=1069.129,437.952,381.705,176.468,36.767,156.939
C03041=1069.139,438.197,381.657,176.476,36.780,156.943
C03042=1069.148,438.442,381.610,176.485,36.793,156.946
C03043=1069.157,438.688,381.562,176.493,36.807,156.950
C03044=1069.165,438.933,381.513,176.502,36.820,156.953
C03045=1069.175,439.178,381.465,176.511,36.833,156.957
C03046=1069.184,439.422,381.417,176.519,36.847,156.960
C03047=1069.193,439.668,381.369,176.529,36.860,156.964
C03048=1069.202,439.913,381.320,176.537,36.874,156.967
C03049=1069.211,440.158,381.272,176.546,36.887,156.971
C03050=1069.220,440.403,381.224,176.555,36.901,156.975
C03051=1069.230,440.648,381.175,176.564,36.914,156.978
C03052=1069.238,440.894,381.127,176.573,36.928,156.982
C03053=1069.247,441.138,381.079,176.582,36.941,156.985
C03054=1069.257,441.383,381.030,176.591,36.955,156.989
C03055=1069.269,441.724,380.962,176.603,36.975,156.994
C03056=1069.283,442.065,380.894,176.616,36.994,156.999
C03057=1069.295,442.407,380.826,176.629,37.013,157.004
C03058=1069.308,442.748,380.757,176.642,37.033,157.010
C03059=1069.318,442.993,380.709,176.651,37.047,157.014
C03060=1069.327,443.238,380.660,176.661,37.061,157.017
C03061=1069.336,443.483,380.611,176.669,37.075,157.021
C03062=1069.345,443.727,380.562,176.679,37.089,157.025
C03063=1069.354,443.973,380.513,176.688,37.103,157.029
C03064=1069.364,444.218,380.464,176.698,37.117,157.032
C03065=1069.373,444.462,380.414,176.708,37.132,157.036
C03066=1069.382,444.707,380.365,176.716,37.146,157.040
C03067=1069.392,444.952,380.316,176.726,37.161,157.044
C03068=1069.402,445.196,380.266,176.736,37.175,157.048
C03069=1069.411,445.442,380.217,176.745,37.190,157.052
C03070=1069.420,445.686,380.167,176.755,37.205,157.056
C03071=1069.430,445.931,380.118,176.765,37.219,157.060
C03072=1069.439,446.175,380.068,176.775,37.233,157.064
C03073=1069.449,446.421,380.019,176.784,37.248,157.068
C03074=1069.458,446.666,379.969,176.794,37.263,157.072
C03075=1069.470,446.961,379.908,176.807,37.281,157.077
C03076=1069.481,447.256,379.848,176.818,37.299,157.082
C03077=1069.493,447.551,379.789,176.831,37.317,157.087
C03078=1069.505,447.846,379.728,176.842,37.335,157.092
C03079=1069.514,448.090,379.679,176.852,37.350,157.096
C03080=1069.525,448.333,379.630,176.862,37.365,157.100
C03081=1069.536,448.578,379.581,176.872,37.379,157.104
C03082=1069.548,448.823,379.532,176.880,37.393,157.107
C03083=1069.562,449.068,379.485,176.889,37.406,157.111
C03084=1069.577,449.312,379.439,176.899,37.419,157.115
C03085=1069.593,449.558,379.393,176.906,37.432,157.118
C03086=1069.610,449.803,379.347,176.915,37.445,157.122
C03087=1069.263,449.804,379.092,176.902,37.581,157.158
C03088=1069.247,449.559,379.138,176.894,37.569,157.155
C03089=1069.230,449.313,379.184,176.885,37.556,157.151
C03090=1069.216,449.068,379.231,176.877,37.544,157.148
C03091=1069.201,448.824,379.278,176.867,37.530,157.144
C03092=1069.189,448.579,379.325,176.858,37.516,157.140
C03093=1069.177,448.334,379.374,176.848,37.502,157.136
C03094=1069.166,448.091,379.424,176.838,37.487,157.132
C03095=1069.156,447.848,379.473,176.828,37.472,157.128
C03096=1069.147,447.603,379.523,176.818,37.457,157.124
C03097=1069.137,447.358,379.573,176.808,37.442,157.120
C03098=1069.128,447.113,379.623,176.797,37.427,157.116
C03099=1069.118,446.869,379.673,176.787,37.413,157.112
C03100=1069.108,446.624,379.722,176.778,37.398,157.108
C03101=1069.099,446.379,379.772,176.768,37.383,157.104
C03102=1069.089,446.134,379.822,176.758,37.368,157.100
C03103=1069.080,445.889,379.872,176.748,37.354,157.096
C03104=1069.070,445.645,379.921,176.738,37.339,157.092
C03105=1069.060,445.400,379.971,176.728,37.325,157.088
C03106=1069.051,445.156,380.021,176.719,37.310,157.084
C03107=1069.042,444.911,380.070,176.710,37.296,157.080
C03108=1069.032,444.666,380.119,176.700,37.281,157.076
C03109=1069.023,444.421,380.169,176.690,37.267,157.072
C03110=1069.014,444.176,380.218,176.681,37.253,157.068
C03111=1069.005,443.931,380.268,176.671,37.239,157.064
C03112=1068.995,443.687,380.317,176.661,37.224,157.061
C03113=1068.986,443.441,380.366,176.652,37.210,157.057
C03114=1068.976,443.196,380.414,176.643,37.196,157.053
C03115=1068.966,442.952,380.464,176.633,37.182,157.049
C03116=1068.953,442.578,380.538,176.619,37.160,157.043
C03117=1068.938,442.205,380.613,176.605,37.140,157.038
C03118=1068.924,441.832,380.687,176.591,37.119,157.032
C03119=1068.910,441.460,380.762,176.577,37.098,157.026
C03120=1068.901,441.215,380.810,176.567,37.084,157.023
C03121=1068.892,440.970,380.859,176.559,37.070,157.019
C03122=1068.882,440.725,380.908,176.550,37.057,157.015
C03123=1068.874,440.480,380.955,176.541,37.043,157.012
C03124=1068.865,440.235,381.005,176.532,37.029,157.008
C03125=1068.855,439.990,381.053,176.522,37.016,157.005
C03126=1068.846,439.745,381.101,176.514,37.002,157.001
C03127=1068.837,439.500,381.150,176.504,36.989,156.997
C03128=1068.824,439.155,381.217,176.492,36.970,156.992
C03129=1068.811,438.811,381.285,176.480,36.951,156.987
C03130=1068.799,438.467,381.353,176.468,36.933,156.982
C03131=1068.786,438.122,381.420,176.456,36.915,156.978
C03132=1068.777,437.877,381.468,176.447,36.901,156.974
C03133=1068.767,437.632,381.516,176.438,36.888,156.971
C03134=1068.758,437.388,381.564,176.430,36.875,156.967
C03135=1068.750,437.142,381.612,176.421,36.862,156.964
C03136=1068.741,436.897,381.659,176.412,36.850,156.961
C03137=1068.731,436.651,381.707,176.404,36.837,156.957
C03138=1068.723,436.406,381.755,176.395,36.824,156.954
C03139=1068.714,436.161,381.802,176.387,36.811,156.950
C03140=1068.704,435.916,381.850,176.379,36.798,156.947
C03141=1068.695,435.671,381.897,176.371,36.785,156.944
C03142=1068.687,435.426,381.945,176.362,36.772,156.940
C03143=1068.678,435.180,381.993,176.354,36.760,156.937
C03144=1068.669,434.935,382.040,176.345,36.748,156.934
C03145=1068.660,434.690,382.087,176.337,36.735,156.930
C03146=1068.652,434.445,382.135,176.328,36.722,156.927
C03147=1068.642,434.199,382.182,176.320,36.710,156.924
C03148=1068.634,433.954,382.229,176.312,36.697,156.921
C03149=1068.625,433.709,382.277,176.304,36.685,156.917
C03150=1068.616,433.463,382.324,176.296,36.672,156.914
C03151=1068.607,433.218,382.371,176.288,36.660,156.911
C03152=1068.599,432.973,382.418,176.280,36.648,156.908
C03153=1068.590,432.727,382.464,176.271,36.635,156.905
C03154=1068.582,432.482,382.512,176.263,36.623,156.902
C03155=1068.574,432.237,382.559,176.255,36.611,156.898
C03156=1068.565,431.991,382.606,176.248,36.599,156.895
C03157=1068.557,431.746,382.653,176.240,36.586,156.892
C03158=1068.548,431.501,382.700,176.232,36.574,156.889
C03159=1068.539,431.255,382.747,176.224,36.562,156.886
C03160=1068.530,431.010,382.793,176.216,36.550,156.883
C03161=1068.521,430.765,382.840,176.208,36.538,156.880
C03162=1068.513,430.519,382.886,176.200,36.526,156.877
C03163=1068.504,430.274,382.933,176.193,36.515,156.874
C03164=1068.496,430.028,382.980,176.185,36.503,156.870
C03165=1068.487,429.782,383.025,176.177,36.491,156.868
C03166=1068.478,429.537,383.072,176.169,36.479,156.864
C03167=1068.470,429.291,383.119,176.162,36.468,156.861
C03168=1068.462,429.065,383.161,176.155,36.457,156.859
C03169=1068.454,428.839,383.204,176.148,36.446,156.856
C03170=1068.446,428.613,383.247,176.140,36.435,156.853
C03171=1068.438,428.387,383.289,176.134,36.425,156.850
C03172=1068.431,428.161,383.332,176.127,36.414,156.848
C03173=1068.423,427.934,383.375,176.120,36.403,156.845
C03174=1068.415,427.708,383.417,176.113,36.393,156.842
C03175=1068.407,427.482,383.460,176.106,36.382,156.840
C03176=1068.399,427.236,383.506,176.099,36.371,156.837
C03177=1068.390,426.990,383.551,176.091,36.359,156.834
C03178=1068.382,426.745,383.598,176.084,36.348,156.831
C03179=1068.373,426.499,383.643,176.076,36.337,156.828
C03180=1068.365,426.253,383.689,176.069,36.326,156.825
C03181=1068.356,426.008,383.735,176.062,36.314,156.822
C03182=1068.348,425.763,383.781,176.054,36.303,156.820
C03183=1068.339,425.517,383.826,176.047,36.292,156.817
C03184=1068.331,425.271,383.872,176.040,36.280,156.814
C03185=1068.322,425.026,383.917,176.032,36.269,156.811
C03186=1068.314,424.780,383.963,176.025,36.258,156.808
C03187=1068.306,424.534,384.008,176.018,36.247,156.805
C03188=1068.298,424.288,384.054,176.011,36.237,156.803
C03189=1068.289,424.043,384.099,176.003,36.226,156.800
C03190=1068.281,423.797,384.145,175.997,36.215,156.797
C03191=1068.273,423.552,384.191,175.989,36.203,156.794
C03192=1068.264,423.306,384.237,175.982,36.193,156.792
C03193=1068.256,423.060,384.281,175.975,36.182,156.789
C03194=1068.248,422.814,384.327,175.968,36.171,156.786
C03195=1068.240,422.569,384.372,175.961,36.160,156.783
C03196=1068.231,422.324,384.417,175.954,36.149,156.781
C03197=1068.223,422.077,384.462,175.947,36.138,156.778
C03198=1068.215,421.832,384.507,175.940,36.128,156.775
C03199=1068.207,421.585,384.553,175.933,36.117,156.773
C03200=1068.199,421.340,384.598,175.926,36.107,156.770
C03201=1068.191,421.094,384.643,175.919,36.096,156.767
C03202=1068.182,420.848,384.688,175.912,36.085,156.765
C03203=1068.174,420.602,384.732,175.906,36.075,156.762
C03204=1068.166,420.357,384.777,175.898,36.064,156.760
C03205=1068.157,420.111,384.822,175.892,36.054,156.757
C03206=1068.150,419.865,384.867,175.884,36.043,156.754
C03207=1068.142,419.619,384.911,175.878,36.033,156.752
C03208=1068.133,419.374,384.956,175.871,36.023,156.749
C03209=1068.125,419.127,385.001,175.864,36.012,156.747
C03210=1068.117,418.882,385.045,175.858,36.002,156.744
C03211=1068.109,418.636,385.090,175.851,35.992,156.742
C03212=1068.101,418.390,385.134,175.844,35.981,156.739
C03213=1068.093,418.143,385.179,175.838,35.971,156.736
C03214=1068.085,417.898,385.224,175.831,35.961,156.734
C03215=1068.076,417.652,385.268,175.825,35.951,156.731
C03216=1068.068,417.406,385.312,175.818,35.941,156.729
C03217=1068.060,417.160,385.357,175.811,35.931,156.726
C03218=1068.052,416.915,385.401,175.805,35.921,156.724
C03219=1068.044,416.669,385.445,175.798,35.910,156.721
C03220=1068.036,416.423,385.490,175.791,35.900,156.719
C03221=1068.028,416.177,385.533,175.785,35.890,156.716
C03222=1068.021,415.931,385.578,175.779,35.880,156.714
C03223=1068.013,415.685,385.623,175.772,35.870,156.712
C03224=1068.005,415.439,385.666,175.765,35.860,156.709
C03225=1067.997,415.193,385.711,175.759,35.851,156.707
C03226=1067.989,414.947,385.755,175.753,35.840,156.704
C03227=1067.981,414.701,385.799,175.747,35.831,156.702
C03228=1067.971,414.414,385.850,175.739,35.820,156.699
C03229=1067.962,414.127,385.901,175.732,35.808,156.696
C03230=1067.953,413.840,385.952,175.724,35.797,156.694
C03231=1067.944,413.554,386.003,175.716,35.785,156.691
C03232=1067.936,413.307,386.047,175.710,35.776,156.688
C03233=1067.928,413.061,386.091,175.704,35.766,156.686
C03234=1067.919,412.815,386.134,175.698,35.756,156.684
C03235=1067.912,412.569,386.178,175.692,35.747,156.682
C03236=1067.904,412.323,386.221,175.685,35.738,156.679
C03237=1067.896,412.077,386.266,175.679,35.728,156.677
C03238=1067.888,411.832,386.308,175.673,35.718,156.674
C03239=1067.880,411.585,386.352,175.667,35.709,156.672
C03240=1067.872,411.339,386.396,175.660,35.699,156.670
C03241=1067.865,411.092,386.439,175.654,35.690,156.668
C03242=1067.856,410.846,386.482,175.648,35.681,156.665
C03243=1067.849,410.601,386.525,175.642,35.671,156.663
C03244=1067.841,410.354,386.569,175.636,35.662,156.661
C03245=1067.833,410.108,386.612,175.630,35.653,156.659
C03246=1067.825,409.863,386.655,175.624,35.643,156.656
C03247=1067.818,409.616,386.699,175.618,35.634,156.654
C03248=1067.809,409.370,386.742,175.611,35.625,156.652
C03249=1067.802,409.124,386.785,175.605,35.615,156.650
C03250=1067.795,408.878,386.828,175.599,35.606,156.647
C03251=1067.786,408.632,386.871,175.593,35.597,156.645
C03252=1067.779,408.386,386.914,175.587,35.588,156.643
C03253=1067.771,408.139,386.957,175.581,35.579,156.641
C03254=1067.764,407.894,387.000,175.575,35.569,156.639
C03255=1067.756,407.647,387.044,175.570,35.561,156.637
C03256=1067.749,407.401,387.086,175.564,35.552,156.634
C03257=1067.740,407.155,387.129,175.558,35.542,156.632
C03258=1067.733,406.908,387.172,175.552,35.533,156.630
C03259=1067.726,406.662,387.215,175.547,35.525,156.628
C03260=1067.718,406.416,387.257,175.541,35.515,156.626
C03261=1067.710,406.170,387.301,175.535,35.506,156.623
C03262=1067.703,405.924,387.343,175.529,35.498,156.621
C03263=1067.695,405.677,387.386,175.523,35.489,156.619
C03264=1067.687,405.432,387.428,175.518,35.480,156.617
C03265=1067.680,405.185,387.471,175.512,35.471,156.615
C03266=1067.672,404.939,387.513,175.506,35.462,156.613
C03267=1067.665,404.692,387.557,175.500,35.453,156.611
C03268=1067.657,404.446,387.599,175.494,35.444,156.609
C03269=1067.649,404.200,387.641,175.489,35.436,156.607
C03270=1067.642,403.953,387.684,175.483,35.427,156.605
C03271=1067.634,403.707,387.726,175.477,35.418,156.603
C03272=1067.627,403.460,387.769,175.471,35.410,156.600
C03273=1067.619,403.215,387.811,175.466,35.401,156.598
C03274=1067.611,402.969,387.853,175.461,35.392,156.596
C03275=1067.603,402.722,387.895,175.455,35.384,156.594
C03276=1067.596,402.476,387.938,175.449,35.375,156.592
C03277=1067.589,402.229,387.979,175.443,35.367,156.590
C03278=1067.581,401.983,388.022,175.438,35.359,156.588
C03279=1067.573,401.737,388.063,175.432,35.350,156.586
C03280=1067.567,401.490,388.106,175.426,35.341,156.584
C03281=1067.559,401.245,388.148,175.421,35.333,156.582
C03282=1067.551,400.998,388.190,175.416,35.325,156.580
C03283=1067.543,400.751,388.232,175.410,35.316,156.578
C03284=1067.535,400.469,388.280,175.404,35.306,156.576
C03285=1067.526,400.186,388.328,175.397,35.297,156.574
C03286=1067.518,399.903,388.376,175.391,35.287,156.572
C03287=1067.509,399.621,388.424,175.385,35.278,156.569
C03288=1067.501,399.375,388.466,175.379,35.270,156.567
C03289=1067.494,399.128,388.507,175.374,35.261,156.565
C03290=1067.487,398.882,388.550,175.369,35.253,156.563
C03291=1067.480,398.635,388.591,175.363,35.245,156.562
C03292=1067.472,398.389,388.633,175.357,35.236,156.560
C03293=1067.465,398.143,388.674,175.353,35.228,156.558
C03294=1067.457,397.897,388.716,175.347,35.220,156.556
C03295=1067.450,397.650,388.757,175.342,35.212,156.554
C03296=1067.442,397.404,388.799,175.336,35.204,156.552
C03297=1067.435,397.158,388.841,175.330,35.196,156.550
C03298=1067.428,396.911,388.882,175.326,35.188,156.548
C03299=1067.420,396.665,388.924,175.320,35.179,156.546
C03300=1067.413,396.418,388.965,175.315,35.172,156.544
C03301=1067.406,396.172,389.006,175.310,35.163,156.543
C03302=1067.398,395.925,389.047,175.304,35.156,156.541
C03303=1067.390,395.680,389.089,175.299,35.148,156.539
C03304=1067.383,395.433,389.130,175.293,35.140,156.537
C03305=1067.376,395.186,389.171,175.289,35.132,156.535
C03306=1067.368,394.940,389.212,175.283,35.124,156.533
C03307=1067.361,394.693,389.254,175.278,35.116,156.531
C03308=1067.354,394.447,389.295,175.272,35.108,156.530
C03309=1067.346,394.200,389.336,175.268,35.100,156.528
C03310=1067.340,393.954,389.377,175.262,35.092,156.526
C03311=1067.332,393.707,389.418,175.257,35.084,156.524
C03312=1067.324,393.461,389.459,175.252,35.077,156.522
C03313=1067.317,393.215,389.500,175.247,35.069,156.521
C03314=1067.310,392.968,389.541,175.241,35.061,156.519
C03315=1067.303,392.722,389.582,175.237,35.054,156.517
C03316=1067.295,392.476,389.623,175.231,35.046,156.515
C03317=1067.288,392.229,389.663,175.226,35.038,156.514
C03318=1067.281,391.982,389.705,175.221,35.030,156.512
C03319=1067.273,391.736,389.745,175.216,35.023,156.510
C03320=1067.266,391.490,389.786,175.210,35.015,156.508
C03321=1067.259,391.243,389.827,175.206,35.007,156.506
C03322=1067.252,390.996,389.868,175.200,34.999,156.505
C03323=1067.244,390.750,389.908,175.195,34.992,156.503
C03324=1067.237,390.503,389.949,175.190,34.984,156.501
C03325=1067.229,390.257,389.989,175.185,34.977,156.499
C03326=1067.222,390.010,390.030,175.181,34.970,156.498
C03327=1067.215,389.764,390.070,175.175,34.962,156.496
C03328=1067.208,389.518,390.111,175.170,34.955,156.494
C03329=1067.200,389.271,390.151,175.165,34.947,156.493
C03330=1067.194,389.024,390.191,175.160,34.940,156.491
C03331=1067.186,388.778,390.232,175.154,34.932,156.489
C03332=1067.179,388.531,390.272,175.150,34.925,156.488
C03333=1067.171,388.285,390.313,175.145,34.918,156.486
C03334=1067.163,388.038,390.353,175.140,34.910,156.484
C03335=1067.157,387.792,390.393,175.135,34.903,156.482
C03336=1067.149,387.545,390.433,175.130,34.895,156.481
C03337=1067.143,387.299,390.474,175.125,34.888,156.479
C03338=1067.135,387.052,390.514,175.120,34.881,156.478
C03339=1067.129,386.805,390.554,175.115,34.873,156.476
C03340=1067.120,386.538,390.597,175.110,34.865,156.474
C03341=1067.112,386.273,390.641,175.105,34.858,156.472
C03342=1067.105,386.006,390.684,175.099,34.850,156.470
C03343=1067.097,385.740,390.727,175.094,34.842,156.469
C03344=1067.090,385.493,390.767,175.089,34.835,156.467
C03345=1067.083,385.246,390.807,175.084,34.828,156.465
C03346=1067.076,384.999,390.847,175.080,34.820,156.464
C03347=1067.069,384.753,390.887,175.074,34.813,156.462
C03348=1067.061,384.506,390.927,175.070,34.806,156.461
C03349=1067.055,384.260,390.967,175.065,34.799,156.459
C03350=1067.047,384.013,391.007,175.060,34.792,156.457
C03351=1067.040,383.766,391.047,175.055,34.785,156.456
C03352=1067.033,383.520,391.087,175.050,34.778,156.454
C03353=1067.026,383.273,391.127,175.046,34.770,156.452
C03354=1067.019,383.026,391.165,175.041,34.764,156.451
C03355=1067.012,382.780,391.206,175.036,34.756,156.449
C03356=1067.005,382.533,391.245,175.031,34.750,156.448
C03357=1066.998,382.287,391.285,175.027,34.742,156.446
C03358=1066.991,382.040,391.325,175.022,34.735,156.445
C03359=1066.984,381.793,391.364,175.017,34.728,156.443
C03360=1066.977,381.546,391.404,175.012,34.721,156.441
C03361=1066.970,381.300,391.444,175.008,34.714,156.440
C03362=1066.963,381.053,391.483,175.003,34.707,156.438
C03363=1066.956,380.806,391.523,174.999,34.701,156.437
C03364=1066.949,380.559,391.562,174.993,34.694,156.435
C03365=1066.942,380.313,391.601,174.989,34.687,156.434
C03366=1066.935,380.066,391.640,174.984,34.680,156.432
C03367=1066.927,379.819,391.680,174.980,34.673,156.431
C03368=1066.920,379.572,391.719,174.974,34.666,156.429
C03369=1066.913,379.326,391.758,174.970,34.660,156.428
C03370=1066.906,379.079,391.798,174.965,34.653,156.426
C03371=1066.899,378.833,391.837,174.961,34.646,156.425
C03372=1066.892,378.586,391.876,174.957,34.639,156.423
C03373=1066.885,378.339,391.915,174.952,34.633,156.422
C03374=1066.878,378.093,391.954,174.947,34.626,156.420
C03375=1066.871,377.846,391.993,174.942,34.619,156.419
C03376=1066.864,377.598,392.032,174.938,34.612,156.417
C03377=1066.857,377.352,392.071,174.933,34.606,156.416
C03378=1066.850,377.105,392.111,174.929,34.599,156.414
C03379=1066.843,376.858,392.150,174.924,34.592,156.413
C03380=1066.836,376.612,392.188,174.920,34.586,156.411
C03381=1066.829,376.365,392.227,174.914,34.579,156.410
C03382=1066.823,376.118,392.266,174.910,34.573,156.408
C03383=1066.816,375.871,392.305,174.906,34.566,156.407
C03384=1066.808,375.624,392.344,174.901,34.559,156.405
C03385=1066.801,375.377,392.384,174.897,34.552,156.404
C03386=1066.795,375.131,392.423,174.892,34.546,156.402
C03387=1066.788,374.884,392.461,174.888,34.539,156.401
C03388=1066.781,374.637,392.500,174.883,34.533,156.399
C03389=1066.774,374.390,392.539,174.879,34.526,156.398
C03390=1066.768,374.143,392.577,174.875,34.520,156.397
C03391=1066.760,373.896,392.615,174.870,34.514,156.395
C03392=1066.753,373.655,392.654,174.866,34.507,156.394
C03393=1066.747,373.414,392.692,174.861,34.501,156.392
C03394=1066.740,373.172,392.729,174.857,34.494,156.391
C03395=1066.734,372.930,392.768,174.853,34.488,156.390
C03396=1066.727,372.688,392.805,174.848,34.481,156.388
C03397=1066.720,372.447,392.843,174.844,34.475,156.387
C03398=1066.714,372.206,392.880,174.839,34.469,156.385
C03399=1066.706,371.964,392.917,174.835,34.463,156.384
C03400=1066.700,371.717,392.956,174.831,34.457,156.383
C03401=1066.693,371.470,392.995,174.826,34.450,156.381
C03402=1066.686,371.223,393.032,174.822,34.444,156.380
C03403=1066.679,370.976,393.071,174.818,34.438,156.379
C03404=1066.671,370.730,393.110,174.813,34.432,156.377
C03405=1066.665,370.482,393.148,174.809,34.425,156.376
C03406=1066.658,370.236,393.187,174.804,34.419,156.374
C03407=1066.651,369.989,393.224,174.800,34.412,156.373
C03408=1066.644,369.742,393.263,174.796,34.406,156.372
C03409=1066.638,369.495,393.301,174.791,34.400,156.370
C03410=1066.630,369.248,393.339,174.787,34.394,156.369
C03411=1066.624,369.001,393.377,174.783,34.387,156.368
C03412=1066.617,368.754,393.415,174.778,34.381,156.366
C03413=1066.610,368.507,393.453,174.774,34.375,156.365
C03414=1066.603,368.260,393.491,174.769,34.369,156.363
C03415=1066.597,368.013,393.529,174.765,34.363,156.362
C03416=1066.590,367.766,393.567,174.761,34.357,156.361
C03417=1066.583,367.519,393.605,174.756,34.351,156.360
C03418=1066.576,367.272,393.643,174.752,34.344,156.358
C03419=1066.569,367.026,393.681,174.748,34.338,156.357
C03420=1066.563,366.778,393.719,174.743,34.332,156.355
C03421=1066.555,366.531,393.757,174.739,34.326,156.354
C03422=1066.549,366.284,393.795,174.735,34.320,156.353
C03423=1066.543,366.037,393.833,174.730,34.314,156.351
C03424=1066.535,365.791,393.871,174.727,34.307,156.350
C03425=1066.529,365.543,393.909,174.723,34.302,156.349
C03426=1066.522,365.297,393.946,174.718,34.295,156.348
C03427=1066.516,365.049,393.984,174.714,34.289,156.346
C03428=1066.509,364.802,394.022,174.710,34.283,156.345
C03429=1066.503,364.555,394.059,174.705,34.277,156.344
C03430=1066.495,364.308,394.097,174.701,34.271,156.342
C03431=1066.488,364.061,394.135,174.697,34.265,156.341
C03432=1066.482,363.814,394.173,174.692,34.259,156.340
C03433=1066.475,363.567,394.210,174.688,34.253,156.338
C03434=1066.468,363.320,394.247,174.685,34.248,156.337
C03435=1066.461,363.073,394.285,174.681,34.241,156.336
C03436=1066.455,362.826,394.322,174.676,34.236,156.335
C03437=1066.448,362.579,394.359,174.672,34.230,156.333
C03438=1066.442,362.332,394.397,174.668,34.224,156.332
C03439=1066.435,362.085,394.435,174.663,34.218,156.331
C03440=1066.427,361.838,394.472,174.659,34.212,156.330
C03441=1066.421,361.590,394.509,174.656,34.206,156.328
C03442=1066.414,361.343,394.546,174.651,34.200,156.327
C03443=1066.408,361.097,394.584,174.647,34.194,156.326
C03444=1066.401,360.849,394.621,174.643,34.189,156.325
C03445=1066.394,360.602,394.658,174.639,34.183,156.323
C03446=1066.387,360.355,394.695,174.634,34.177,156.322
C03447=1066.381,360.107,394.733,174.631,34.171,156.321
C03448=1066.374,359.875,394.767,174.627,34.166,156.320
C03449=1066.368,359.642,394.803,174.622,34.160,156.318
C03450=1066.362,359.409,394.838,174.619,34.155,156.317
C03451=1066.355,359.177,394.873,174.615,34.149,156.316
C03452=1066.349,358.944,394.908,174.612,34.144,156.315
C03453=1066.343,358.710,394.943,174.607,34.138,156.314
C03454=1066.336,358.478,394.977,174.603,34.133,156.313
C03455=1066.330,358.245,395.012,174.600,34.128,156.312
C03456=1066.324,357.997,395.049,174.596,34.122,156.310
C03457=1066.317,357.751,395.086,174.591,34.116,156.309
C03458=1066.310,357.503,395.123,174.587,34.111,156.308
C03459=1066.303,357.257,395.160,174.584,34.105,156.307
C03460=1066.296,357.009,395.197,174.580,34.099,156.305
C03461=1066.290,356.762,395.234,174.575,34.094,156.304
C03462=1066.283,356.514,395.270,174.571,34.088,156.303
C03463=1066.276,356.268,395.308,174.568,34.083,156.302
C03464=1066.269,356.020,395.344,174.564,34.077,156.301
C03465=1066.263,355.773,395.381,174.559,34.071,156.299
C03466=1066.257,355.526,395.417,174.555,34.066,156.298
C03467=1066.250,355.279,395.455,174.552,34.060,156.297
C03468=1066.243,355.032,395.491,174.548,34.054,156.296
C03469=1066.236,354.784,395.528,174.543,34.049,156.295
C03470=1066.230,354.537,395.564,174.539,34.043,156.294
C03471=1066.224,354.290,395.601,174.536,34.038,156.292
C03472=1066.217,354.042,395.638,174.532,34.032,156.291
C03473=1066.210,353.795,395.674,174.527,34.027,156.290
C03474=1066.204,353.548,395.711,174.524,34.021,156.289
C03475=1066.197,353.300,395.747,174.520,34.016,156.288
C03476=1066.191,353.053,395.784,174.516,34.010,156.287
C03477=1066.184,352.806,395.820,174.511,34.004,156.285
C03478=1066.177,352.559,395.856,174.508,33.999,156.284
C03479=1066.170,352.312,395.893,174.504,33.993,156.283
C03480=1066.164,352.064,395.929,174.500,33.988,156.282
C03481=1066.158,351.817,395.966,174.497,33.982,156.281
C03482=1066.151,351.570,396.003,174.492,33.977,156.280
C03483=1066.144,351.323,396.039,174.488,33.972,156.279
C03484=1066.137,351.076,396.075,174.485,33.966,156.277
C03485=1066.131,350.829,396.111,174.481,33.961,156.276
C03486=1066.124,350.580,396.148,174.476,33.956,156.275
C03487=1066.117,350.334,396.183,174.473,33.950,156.274
C03488=1066.111,350.087,396.220,174.469,33.945,156.273
C03489=1066.105,349.840,396.256,174.465,33.939,156.272
C03490=1066.098,349.591,396.292,174.462,33.934,156.271
C03491=1066.091,349.344,396.328,174.457,33.928,156.269
C03492=1066.085,349.097,396.365,174.453,33.923,156.268
C03493=1066.079,348.850,396.400,174.450,33.918,156.267
C03494=1066.072,348.603,396.436,174.446,33.912,156.266
C03495=1066.065,348.355,396.472,174.442,33.907,156.265
C03496=1066.059,348.108,396.509,174.438,33.902,156.264
C03497=1066.051,347.861,396.545,174.434,33.896,156.263
C03498=1066.045,347.613,396.580,174.431,33.891,156.262
C03499=1066.039,347.366,396.617,174.427,33.886,156.261
C03500=1066.032,347.119,396.652,174.423,33.880,156.259
C03501=1066.026,346.872,396.688,174.419,33.875,156.258
C03502=1066.020,346.624,396.724,174.415,33.870,156.257
C03503=1066.012,346.377,396.760,174.412,33.865,156.256
C03504=1066.006,346.146,396.794,174.408,33.860,156.255
C03505=1066.001,345.915,396.827,174.405,33.855,156.254
C03506=1065.995,345.684,396.860,174.400,33.850,156.253
C03507=1065.989,345.453,396.893,174.397,33.845,156.252
C03508=1065.983,345.222,396.927,174.394,33.840,156.251
C03509=1065.976,344.991,396.961,174.390,33.835,156.250
C03510=1065.970,344.761,396.994,174.387,33.830,156.249
C03511=1065.964,344.530,397.027,174.384,33.826,156.248
C03512=1065.958,344.282,397.063,174.379,33.820,156.247
C03513=1065.951,344.035,397.098,174.376,33.815,156.246
C03514=1065.945,343.787,397.134,174.372,33.810,156.245
C03515=1065.938,343.541,397.169,174.369,33.805,156.244
C03516=1065.932,343.293,397.205,174.365,33.799,156.243
C03517=1065.925,343.046,397.240,174.361,33.795,156.242
C03518=1065.919,342.798,397.275,174.357,33.789,156.241
C03519=1065.913,342.550,397.311,174.353,33.784,156.239
C03520=1065.906,342.303,397.346,174.350,33.779,156.238
C03521=1065.900,342.055,397.382,174.346,33.774,156.237
C03522=1065.893,341.808,397.417,174.343,33.769,156.236
C03523=1065.886,341.561,397.453,174.339,33.764,156.235
C03524=1065.880,341.314,397.489,174.335,33.759,156.234
C03525=1065.873,341.066,397.524,174.331,33.754,156.233
C03526=1065.866,340.819,397.559,174.328,33.749,156.232
C03527=1065.860,340.571,397.595,174.324,33.743,156.231
C03528=1065.854,340.324,397.630,174.321,33.739,156.230
C03529=1065.847,340.076,397.664,174.317,33.733,156.229
C03530=1065.840,339.829,397.699,174.313,33.728,156.228
C03531=1065.834,339.581,397.735,174.309,33.723,156.227
C03532=1065.827,339.334,397.770,174.306,33.718,156.226
C03533=1065.821,339.086,397.805,174.302,33.713,156.225
C03534=1065.815,338.839,397.841,174.299,33.708,156.224
C03535=1065.809,338.592,397.876,174.295,33.703,156.223
C03536=1065.802,338.344,397.911,174.292,33.698,156.222
C03537=1065.796,338.096,397.946,174.287,33.693,156.221
C03538=1065.789,337.849,397.981,174.284,33.688,156.220
C03539=1065.782,337.601,398.016,174.280,33.683,156.219
C03540=1065.776,337.355,398.051,174.277,33.678,156.218
C03541=1065.770,337.107,398.086,174.273,33.673,156.217
C03542=1065.764,336.859,398.121,174.270,33.668,156.216
C03543=1065.757,336.612,398.156,174.266,33.663,156.215
C03544=1065.751,336.364,398.191,174.262,33.658,156.214
C03545=1065.744,336.116,398.226,174.258,33.653,156.213
C03546=1065.738,335.870,398.261,174.255,33.648,156.212
C03547=1065.731,335.622,398.295,174.252,33.644,156.211
C03548=1065.724,335.374,398.330,174.248,33.639,156.210
C03549=1065.718,335.126,398.365,174.245,33.634,156.209
C03550=1065.711,334.879,398.400,174.241,33.629,156.208
C03551=1065.705,334.632,398.434,174.238,33.624,156.207
C03552=1065.699,334.384,398.469,174.233,33.619,156.206
C03553=1065.692,334.136,398.503,174.230,33.614,156.205
C03554=1065.685,333.889,398.539,174.227,33.609,156.204
C03555=1065.679,333.642,398.573,174.223,33.604,156.203
C03556=1065.673,333.394,398.608,174.220,33.600,156.202
C03557=1065.666,333.146,398.642,174.216,33.595,156.201
C03558=1065.660,332.899,398.676,174.213,33.590,156.200
C03559=1065.654,332.652,398.711,174.210,33.585,156.199
C03560=1065.648,332.418,398.745,174.205,33.580,156.198
C03561=1065.642,332.185,398.777,174.202,33.576,156.197
C03562=1065.636,331.951,398.809,174.199,33.571,156.196
C03563=1065.630,331.719,398.842,174.196,33.567,156.195
C03564=1065.624,331.485,398.874,174.193,33.562,156.194
C03565=1065.618,331.251,398.907,174.189,33.558,156.193
C03566=1065.612,331.018,398.940,174.186,33.553,156.192
C03567=1065.606,330.784,398.971,174.183,33.548,156.191
C03568=1065.600,330.538,399.006,174.180,33.544,156.190
C03569=1065.593,330.290,399.040,174.175,33.539,156.189
C03570=1065.586,330.042,399.074,174.172,33.534,156.188
C03571=1065.580,329.794,399.109,174.169,33.530,156.188
C03572=1065.573,329.547,399.142,174.165,33.525,156.187
C03573=1065.567,329.299,399.177,174.162,33.521,156.186
C03574=1065.560,329.051,399.211,174.158,33.516,156.185
C03575=1065.553,328.804,399.245,174.155,33.511,156.184
C03576=1065.547,328.556,399.279,174.152,33.507,156.183
C03577=1065.541,328.309,399.313,174.148,33.502,156.182
C03578=1065.534,328.062,399.348,174.145,33.497,156.181
C03579=1065.528,327.813,399.381,174.141,33.492,156.180
C03580=1065.521,327.566,399.415,174.137,33.488,156.179
C03581=1065.514,327.318,399.449,174.134,33.483,156.178
C03582=1065.509,327.071,399.483,174.131,33.479,156.177
C03583=1065.501,326.823,399.517,174.127,33.474,156.176
C03584=1065.495,326.575,399.552,174.124,33.469,156.175
C03585=1065.488,326.328,399.585,174.121,33.464,156.174
C03586=1065.482,326.080,399.619,174.117,33.460,156.174
C03587=1065.476,325.833,399.653,174.114,33.455,156.173
C03588=1065.469,325.585,399.687,174.111,33.451,156.172
C03589=1065.463,325.338,399.721,174.107,33.446,156.171
C03590=1065.456,325.090,399.754,174.103,33.441,156.170
C03591=1065.450,324.843,399.789,174.100,33.437,156.169
C03592=1065.444,324.595,399.823,174.096,33.432,156.168
C03593=1065.437,324.348,399.856,174.093,33.428,156.167
C03594=1065.431,324.099,399.890,174.090,33.423,156.166
C03595=1065.424,323.852,399.924,174.087,33.418,156.165
C03596=1065.418,323.604,399.958,174.083,33.413,156.164
C03597=1065.411,323.357,399.991,174.080,33.409,156.163
C03598=1065.406,323.109,400.025,174.077,33.405,156.163
C03599=1065.399,322.862,400.059,174.074,33.400,156.162
C03600=1065.393,322.614,400.093,174.070,33.395,156.161
C03601=1065.387,322.366,400.126,174.067,33.391,156.160
C03602=1065.380,322.119,400.160,174.063,33.386,156.159
C03603=1065.374,321.871,400.193,174.060,33.381,156.158
C03604=1065.367,321.623,400.227,174.056,33.377,156.157
C03605=1065.362,321.375,400.260,174.053,33.372,156.156
C03606=1065.354,321.128,400.294,174.050,33.368,156.155
C03607=1065.349,320.880,400.328,174.047,33.363,156.154
C03608=1065.342,320.633,400.361,174.043,33.359,156.153
C03609=1065.336,320.385,400.395,174.040,33.354,156.152
C03610=1065.330,320.137,400.428,174.037,33.349,156.152
C03611=1065.324,319.890,400.462,174.034,33.345,156.151
C03612=1065.317,319.642,400.495,174.030,33.340,156.150
C03613=1065.311,319.394,400.529,174.027,33.336,156.149
C03614=1065.305,319.147,400.562,174.024,33.331,156.148
C03615=1065.299,318.899,400.595,174.021,33.327,156.147
C03616=1065.292,318.662,400.628,174.017,33.323,156.146
C03617=1065.287,318.426,400.659,174.014,33.318,156.145
C03618=1065.281,318.190,400.691,174.011,33.314,156.144
C03619=1065.274,317.954,400.723,174.008,33.309,156.144
C03620=1065.269,317.718,400.754,174.005,33.305,156.143
C03621=1065.263,317.481,400.787,174.001,33.300,156.142
C03622=1065.257,317.245,400.819,173.998,33.296,156.141
C03623=1065.251,317.009,400.850,173.995,33.292,156.140
C03624=1065.245,316.761,400.883,173.992,33.287,156.139
C03625=1065.239,316.513,400.917,173.989,33.283,156.138
C03626=1065.232,316.266,400.950,173.986,33.278,156.137
C03627=1065.227,316.018,400.983,173.983,33.274,156.137
C03628=1065.221,315.770,401.016,173.980,33.270,156.136
C03629=1065.214,315.523,401.049,173.976,33.265,156.135
C03630=1065.209,315.275,401.082,173.973,33.260,156.134
C03631=1065.202,315.027,401.115,173.970,33.256,156.133
C03632=1065.196,314.779,401.149,173.967,33.252,156.132
C03633=1065.190,314.532,401.182,173.964,33.247,156.131
C03634=1065.183,314.284,401.215,173.960,33.243,156.130
C03635=1065.178,314.036,401.248,173.957,33.238,156.129
C03636=1065.172,313.788,401.281,173.953,33.234,156.129
C03637=1065.165,313.541,401.314,173.950,33.229,156.128
